// TIA Portal V17 export
// export: Created 2023-11-13T12:30:02.9222123Z, ExportSetting WithDefaults, DisplayName Totally Integrated Automation Portal, DisplayVersion V17, DisplayName TIA Portal Openness, DisplayVersion V17, DisplayName TIA Portal Version Control Interface, DisplayVersion V17, DisplayName STEP 7 Professional, DisplayVersion V17, DisplayName STEP 7 Safety, DisplayVersion V17, DisplayName WinCC Professional, DisplayVersion V17
FUNCTION_BLOCK "Motor"   // FB11, FBD
{ S7_Optimized_Access := 'TRUE' }
VERSION : 0.1
// stored: AutoNumber true, IsIECCheckEnabled false, IsRetainMemResEnabled false, MemoryReserve 100, SetENOAutomatically false, UDAEnableTagReadback false
   VAR_INPUT
      CON : Bool;
      COFF : Bool := 1;
      TagName : String[16];
      "PCS/PLC" : Bool;
      PCS_Auto : Bool;
      Ready : Bool;
      Running : Bool;
      STAITL : Bool := 1;
      PSTITL : Bool := 1;
      STPITL : Bool := 1;
      OPITL : Bool := 1;
      PRTITL : Bool := 1;
      FO { ExternalAccessible := 'False'; ExternalVisible := 'False'; ExternalWritable := 'False'} : Bool;   // First Out
      PHYFB : Bool := 1;
   END_VAR
   VAR_OUTPUT
      AVBL : Bool;
      ON : Bool;
      RUN : Bool;
      Start_PCS : Bool;
      Stop_PCS : Bool;
      Interlock_PCS : Bool;
      Screen : Bool;
   END_VAR
   VAR_IN_OUT
      Popup : "Popup_MtrOnOff";   // Common Popup Data
   END_VAR
   VAR
      "Local start" : Bool;
      "Local stop" : Bool;
      Remote : Bool;
      "Remote release" : Bool;
      Local : Bool;
      "Local release" : Bool;
      "Motor fault (electrically)" : Bool;
      "Feedback contactor" : Bool;
      Start : Bool;
      Stop : Bool;
      FDBCK : Bool;
      "Stop/ITL" : Bool;
      "Stop/Run" : Bool;
      IEC_Timer_Feedback_On { S7_SetPoint := 'True'} : TON_TIME;
      IEC_Timer_Feedback_Off { S7_SetPoint := 'True'} : TON_TIME;
      IEC_Timer_Feedback_Run { S7_SetPoint := 'True'} : TON_TIME;
      FDBCK_On { S7_SetPoint := 'True'} : Bool;
      FDBCK_Off { S7_SetPoint := 'True'} : Bool;
      FDBCK_Run { S7_SetPoint := 'True'} : Bool;
   END_VAR
   VAR RETAIN
      Param { ExternalAccessible := 'False'; ExternalVisible := 'False'; ExternalWritable := 'False'} : Struct   // Internal Parameters
         ReversingMotor { ExternalAccessible := 'False'; ExternalVisible := 'False'; ExternalWritable := 'False'; S7_SetPoint := 'True'} : Bool := False;   // 1:Enable Direction Select
         SpeedSelect { ExternalAccessible := 'False'; ExternalVisible := 'False'; ExternalWritable := 'False'; S7_SetPoint := 'True'} : Bool := False;   // 1:Enable Speed Select
         EN_FB_Forward { ExternalAccessible := 'False'; ExternalVisible := 'False'; ExternalWritable := 'False'; S7_SetPoint := 'True'} : Bool := true;   // 1:Enable FB_Forward
         EN_FB_Revsere { ExternalAccessible := 'False'; ExternalVisible := 'False'; ExternalWritable := 'False'; S7_SetPoint := 'True'} : Bool := true;   // 1:Enable FB_Reverse
         Disable_MCC_FLT { ExternalAccessible := 'False'; ExternalVisible := 'False'; ExternalWritable := 'False'; S7_SetPoint := 'True'} : Bool := false;   // 1:Disable MCC_FLT
         Disable_StartFLT { ExternalAccessible := 'False'; ExternalVisible := 'False'; ExternalWritable := 'False'; S7_SetPoint := 'True'} : Bool := false;   // 1:Disable StartFLT
         Disable_StopFLT { ExternalAccessible := 'False'; ExternalVisible := 'False'; ExternalWritable := 'False'; S7_SetPoint := 'True'} : Bool := false;   // 1:Disable StopFLT
         Disable_ForwardFLT { ExternalAccessible := 'False'; ExternalVisible := 'False'; ExternalWritable := 'False'; S7_SetPoint := 'True'} : Bool := false;   // 1:Disable ForwardFLT
         Disable_ReverseFLT { ExternalAccessible := 'False'; ExternalVisible := 'False'; ExternalWritable := 'False'; S7_SetPoint := 'True'} : Bool := false;   // 1:Disable ReverseFLT
         CMD_PulseWidth { ExternalAccessible := 'False'; ExternalVisible := 'False'; ExternalWritable := 'False'; S7_SetPoint := 'True'} : Time := t#2s;   // Command Pulse width
         WatchdogTime { ExternalAccessible := 'False'; ExternalVisible := 'False'; ExternalWritable := 'False'; S7_SetPoint := 'True'} : Array[0..5] of Real;   // Watchdog time for Fault detection
         Bumpless { ExternalAccessible := 'False'; ExternalVisible := 'False'; ExternalWritable := 'False'; S7_SetPoint := 'True'} : Bool := true;   // 1:Bumpless Switching to PLC Remote
         OpeBy2Step { ExternalAccessible := 'False'; ExternalVisible := 'False'; ExternalWritable := 'False'; S7_SetPoint := 'True'} : Bool := true;   // 1:2Step Operation
         PopupTime { ExternalAccessible := 'False'; ExternalVisible := 'False'; ExternalWritable := 'False'; S7_SetPoint := 'True'} : Time := T#60s;   // Time to close Confiramtion box
         TotalNoOfHMI { ExternalAccessible := 'False'; ExternalVisible := 'False'; ExternalWritable := 'False'; S7_SetPoint := 'True'} : Int := 1;   // Total Number of HMI
      END_STRUCT;
   END_VAR
   VAR
      icon : "icon_MtrOnOff";   // Icon Data
      HMI : "Popup_MtrOnOff";   // HMI Display Data
      ActiveHMI { ExternalAccessible := 'False'; ExternalVisible := 'False'; ExternalWritable := 'False'} : "Popup_MtrOnOff";   // Active HMI Data (Work Data)
      PassiveHMI { ExternalAccessible := 'False'; ExternalVisible := 'False'; ExternalWritable := 'False'} : "Popup_MtrOnOff";   // Passive HMI Object Code
      PopupCtrl { ExternalAccessible := 'False'; ExternalVisible := 'False'; ExternalWritable := 'False'} : Struct   // Popup Control Data
         Opened { ExternalAccessible := 'False'; ExternalVisible := 'False'; ExternalWritable := 'False'} : Bool;   // Popup is opened on the HMI
         Activate { ExternalAccessible := 'False'; ExternalVisible := 'False'; ExternalWritable := 'False'} : Bool;   // Any Operating on the HMI
         ValueChange { ExternalAccessible := 'False'; ExternalVisible := 'False'; ExternalWritable := 'False'} : Bool;   // Any Value is chaging on the HMI
         OperationBlocked { ExternalAccessible := 'False'; ExternalVisible := 'False'; ExternalWritable := 'False'} : Bool;   // Operation is blocked (inhibited)
         TagNameNotSame { ExternalAccessible := 'False'; ExternalVisible := 'False'; ExternalWritable := 'False'} : Bool;   // Tag name is not same with opened Popup on the HMI
      END_STRUCT;
      Modifying { ExternalAccessible := 'False'; ExternalVisible := 'False'; ExternalWritable := 'False'} : Struct   // Value is being modifyed on HMI
         AnyValue { ExternalAccessible := 'False'; ExternalVisible := 'False'; ExternalWritable := 'False'} : Bool;
         WatchdogTime_MccFLT { ExternalAccessible := 'False'; ExternalVisible := 'False'; ExternalWritable := 'False'} : Bool;
         WatchdogTime_StartFLT { ExternalAccessible := 'False'; ExternalVisible := 'False'; ExternalWritable := 'False'; S7_SetPoint := 'True'} : Bool;
         WatchdogTime_StopFLT { ExternalAccessible := 'False'; ExternalVisible := 'False'; ExternalWritable := 'False'; S7_SetPoint := 'True'} : Bool;
         WatchdogTime_ForwardFLT { ExternalAccessible := 'False'; ExternalVisible := 'False'; ExternalWritable := 'False'; S7_SetPoint := 'True'} : Bool;
         WatchdogTime_ReverseFLT { ExternalAccessible := 'False'; ExternalVisible := 'False'; ExternalWritable := 'False'; S7_SetPoint := 'True'} : Bool;
      END_STRUCT;
      previous { ExternalAccessible := 'False'; ExternalVisible := 'False'; ExternalWritable := 'False'} : Struct   // Previous Values
         WatchdogTime { ExternalAccessible := 'False'; ExternalVisible := 'False'; ExternalWritable := 'False'} : Array[0..5] of Real;
      END_STRUCT;
      Check { ExternalAccessible := 'False'; ExternalVisible := 'False'; ExternalWritable := 'False'} : Struct   // Check Value
         PBNo { ExternalAccessible := 'False'; ExternalVisible := 'False'; ExternalWritable := 'False'} : Int;
         WatchdogTime { ExternalAccessible := 'False'; ExternalVisible := 'False'; ExternalWritable := 'False'} : Real;
      END_STRUCT;
      HMI_PB { ExternalAccessible := 'False'; ExternalVisible := 'False'; ExternalWritable := 'False'} : Struct   // Push Buttons on Popup
         Remote { ExternalAccessible := 'False'; ExternalVisible := 'False'; ExternalWritable := 'False'} : Bool;
         Local { ExternalAccessible := 'False'; ExternalVisible := 'False'; ExternalWritable := 'False'} : Bool;
         Auto { ExternalAccessible := 'False'; ExternalVisible := 'False'; ExternalWritable := 'False'} : Bool;
         Manual { ExternalAccessible := 'False'; ExternalVisible := 'False'; ExternalWritable := 'False'} : Bool;
         Forward { ExternalAccessible := 'False'; ExternalVisible := 'False'; ExternalWritable := 'False'} : Bool;
         Reverse { ExternalAccessible := 'False'; ExternalVisible := 'False'; ExternalWritable := 'False'} : Bool;
         Speed1 { ExternalAccessible := 'False'; ExternalVisible := 'False'; ExternalWritable := 'False'} : Bool;
         Speed2 { ExternalAccessible := 'False'; ExternalVisible := 'False'; ExternalWritable := 'False'} : Bool;
         Start { ExternalAccessible := 'False'; ExternalVisible := 'False'; ExternalWritable := 'False'} : Bool;
         Stop { ExternalAccessible := 'False'; ExternalVisible := 'False'; ExternalWritable := 'False'} : Bool;
         ResetRT { ExternalAccessible := 'False'; ExternalVisible := 'False'; ExternalWritable := 'False'} : Bool;
         FO { ExternalAccessible := 'False'; ExternalVisible := 'False'; ExternalWritable := 'False'} : Bool;
      END_STRUCT;
      PLC_IN { ExternalAccessible := 'False'; ExternalVisible := 'False'; ExternalWritable := 'False'} : Struct   // PLC Signal operated on HMI
         Remote { ExternalAccessible := 'False'; ExternalVisible := 'False'; ExternalWritable := 'False'} : Bool;   // 0:Local / 1:Remote by PLC(HMI)
         Auto { ExternalAccessible := 'False'; ExternalVisible := 'False'; ExternalWritable := 'False'} : Bool;   // 0:Manual / 1:Auto by PLC(HMI)
         Start { ExternalAccessible := 'False'; ExternalVisible := 'False'; ExternalWritable := 'False'} : Bool;   // 1:Start by PLC(HMI)
         Stop { ExternalAccessible := 'False'; ExternalVisible := 'False'; ExternalWritable := 'False'} : Bool;   // 1: Stop by PLC(HMI)
         Reverse { ExternalAccessible := 'False'; ExternalVisible := 'False'; ExternalWritable := 'False'} : Bool;   // 0:Forward / 1:Reverse by PLC(HMI)
         Speed { ExternalAccessible := 'False'; ExternalVisible := 'False'; ExternalWritable := 'False'} : Bool;   // 0:Speed1 / 1:Speed2 by PLC(HMI)
      END_STRUCT;
      PBNo { ExternalAccessible := 'False'; ExternalVisible := 'False'; ExternalWritable := 'False'} : Int;   // Internal PBNo
      HMI_Operating { ExternalAccessible := 'False'; ExternalVisible := 'False'; ExternalWritable := 'False'} : Bool;   // Operating on HMI
      Popup_Open { ExternalAccessible := 'False'; ExternalVisible := 'False'; ExternalWritable := 'False'} : Bool;   // Any Popup is Opened
      Popup_Activate { ExternalAccessible := 'False'; ExternalVisible := 'False'; ExternalWritable := 'False'} : Bool;   // Any Popup is Activated
      Init { ExternalAccessible := 'False'; ExternalVisible := 'False'; ExternalWritable := 'False'} : Bool;
      ExternalReset { ExternalAccessible := 'False'; ExternalVisible := 'False'; ExternalWritable := 'False'} : Bool;   // External Reset
      Confirm { ExternalAccessible := 'False'; ExternalVisible := 'False'; ExternalWritable := 'False'} : Bool;   // Confirm Action
      Cancel { ExternalAccessible := 'False'; ExternalVisible := 'False'; ExternalWritable := 'False'} : Bool;   // Cancel Action
      CancelTimer { ExternalAccessible := 'False'; ExternalVisible := 'False'; ExternalWritable := 'False'} : Bool;   // Cancel Timer
      Enable { ExternalAccessible := 'False'; ExternalVisible := 'False'; ExternalWritable := 'False'} : Bool;   // 1:Enable Motor Operation
      Start_1 { ExternalAccessible := 'False'; ExternalVisible := 'False'; ExternalWritable := 'False'} : Bool;   // 1:Start Command ON
      Field_ForwardPLS { ExternalAccessible := 'False'; ExternalVisible := 'False'; ExternalWritable := 'False'} : Bool;   // Field Forward Pulse
      Field_ReversePLS { ExternalAccessible := 'False'; ExternalVisible := 'False'; ExternalWritable := 'False'} : Bool;   // Field Reverse Pulse
      SIM { ExternalAccessible := 'False'; ExternalVisible := 'False'; ExternalWritable := 'False'} : Bool;   // 1: SIM Mode (Automatic Answer)
      RT { ExternalAccessible := 'False'; ExternalVisible := 'False'; ExternalWritable := 'False'} : Struct   // RunTime
         hour { ExternalAccessible := 'False'; ExternalVisible := 'False'; ExternalWritable := 'False'} : DInt;
         min { ExternalAccessible := 'False'; ExternalVisible := 'False'; ExternalWritable := 'False'} : DInt;
         sec { ExternalAccessible := 'False'; ExternalVisible := 'False'; ExternalWritable := 'False'} : Int;
         ActSec { ExternalAccessible := 'False'; ExternalVisible := 'False'; ExternalWritable := 'False'} : USInt;
         Edge { ExternalAccessible := 'False'; ExternalVisible := 'False'; ExternalWritable := 'False'} : Bool;
         Reset { ExternalAccessible := 'False'; ExternalVisible := 'False'; ExternalWritable := 'False'} : Bool;
      END_STRUCT;
      Clear { ExternalAccessible := 'False'; ExternalVisible := 'False'; ExternalWritable := 'False'} : "Popup_MtrOnOff";   // for Clear Popup Data
      Edge { ExternalAccessible := 'False'; ExternalVisible := 'False'; ExternalWritable := 'False'} : Struct   // for Edging
         Remote { ExternalAccessible := 'False'; ExternalVisible := 'False'; ExternalWritable := 'False'} : Bool;
         Local { ExternalAccessible := 'False'; ExternalVisible := 'False'; ExternalWritable := 'False'} : Bool;
         Auto { ExternalAccessible := 'False'; ExternalVisible := 'False'; ExternalWritable := 'False'} : Bool;
         Manual { ExternalAccessible := 'False'; ExternalVisible := 'False'; ExternalWritable := 'False'} : Bool;
         Forward { ExternalAccessible := 'False'; ExternalVisible := 'False'; ExternalWritable := 'False'} : Bool;
         Reverse { ExternalAccessible := 'False'; ExternalVisible := 'False'; ExternalWritable := 'False'} : Bool;
         Speed1 { ExternalAccessible := 'False'; ExternalVisible := 'False'; ExternalWritable := 'False'} : Bool;
         Speed2 { ExternalAccessible := 'False'; ExternalVisible := 'False'; ExternalWritable := 'False'} : Bool;
         Start { ExternalAccessible := 'False'; ExternalVisible := 'False'; ExternalWritable := 'False'} : Bool;
         Stop { ExternalAccessible := 'False'; ExternalVisible := 'False'; ExternalWritable := 'False'} : Bool;
         HMI_Remote { ExternalAccessible := 'False'; ExternalVisible := 'False'; ExternalWritable := 'False'} : Bool;
         HMI_Local { ExternalAccessible := 'False'; ExternalVisible := 'False'; ExternalWritable := 'False'} : Bool;
         HMI_Auto { ExternalAccessible := 'False'; ExternalVisible := 'False'; ExternalWritable := 'False'} : Bool;
         HMI_Manual { ExternalAccessible := 'False'; ExternalVisible := 'False'; ExternalWritable := 'False'} : Bool;
         HMI_Forward { ExternalAccessible := 'False'; ExternalVisible := 'False'; ExternalWritable := 'False'} : Bool;
         HMI_Reverse { ExternalAccessible := 'False'; ExternalVisible := 'False'; ExternalWritable := 'False'} : Bool;
         HMI_Speed1 { ExternalAccessible := 'False'; ExternalVisible := 'False'; ExternalWritable := 'False'} : Bool;
         HMI_Speed2 { ExternalAccessible := 'False'; ExternalVisible := 'False'; ExternalWritable := 'False'} : Bool;
         PCS_Remote { ExternalAccessible := 'False'; ExternalVisible := 'False'; ExternalWritable := 'False'} : Bool;
         PCS_Local { ExternalAccessible := 'False'; ExternalVisible := 'False'; ExternalWritable := 'False'} : Bool;
         PCS_Auto { ExternalAccessible := 'False'; ExternalVisible := 'False'; ExternalWritable := 'False'} : Bool;
         PCS_Manual { ExternalAccessible := 'False'; ExternalVisible := 'False'; ExternalWritable := 'False'} : Bool;
         PCS_Forward { ExternalAccessible := 'False'; ExternalVisible := 'False'; ExternalWritable := 'False'} : Bool;
         PCS_Reverse { ExternalAccessible := 'False'; ExternalVisible := 'False'; ExternalWritable := 'False'} : Bool;
         PCS_Speed1 { ExternalAccessible := 'False'; ExternalVisible := 'False'; ExternalWritable := 'False'} : Bool;
         PCS_Speed2 { ExternalAccessible := 'False'; ExternalVisible := 'False'; ExternalWritable := 'False'} : Bool;
         PCS_Start { ExternalAccessible := 'False'; ExternalVisible := 'False'; ExternalWritable := 'False'} : Bool;
         PCS_Stop { ExternalAccessible := 'False'; ExternalVisible := 'False'; ExternalWritable := 'False'} : Bool;
         PLC_Remote { ExternalAccessible := 'False'; ExternalVisible := 'False'; ExternalWritable := 'False'} : Bool;
         PLC_Local { ExternalAccessible := 'False'; ExternalVisible := 'False'; ExternalWritable := 'False'} : Bool;
         PLC_Auto { ExternalAccessible := 'False'; ExternalVisible := 'False'; ExternalWritable := 'False'} : Bool;
         PLC_Manual { ExternalAccessible := 'False'; ExternalVisible := 'False'; ExternalWritable := 'False'} : Bool;
         PLC_Forward { ExternalAccessible := 'False'; ExternalVisible := 'False'; ExternalWritable := 'False'} : Bool;
         PLC_Reverse { ExternalAccessible := 'False'; ExternalVisible := 'False'; ExternalWritable := 'False'} : Bool;
         PLC_Speed1 { ExternalAccessible := 'False'; ExternalVisible := 'False'; ExternalWritable := 'False'} : Bool;
         PLC_Speed2 { ExternalAccessible := 'False'; ExternalVisible := 'False'; ExternalWritable := 'False'} : Bool;
         PLC_Start { ExternalAccessible := 'False'; ExternalVisible := 'False'; ExternalWritable := 'False'} : Bool;
         PLC_Stop { ExternalAccessible := 'False'; ExternalVisible := 'False'; ExternalWritable := 'False'} : Bool;
         Auto_Start { ExternalAccessible := 'False'; ExternalVisible := 'False'; ExternalWritable := 'False'} : Bool;
         Auto_Stop { ExternalAccessible := 'False'; ExternalVisible := 'False'; ExternalWritable := 'False'} : Bool;
         Auto_Forward { ExternalAccessible := 'False'; ExternalVisible := 'False'; ExternalWritable := 'False'} : Bool;
         Auto_Reverse { ExternalAccessible := 'False'; ExternalVisible := 'False'; ExternalWritable := 'False'} : Bool;
         Auto_Speed1 { ExternalAccessible := 'False'; ExternalVisible := 'False'; ExternalWritable := 'False'} : Bool;
         Auto_Speed2 { ExternalAccessible := 'False'; ExternalVisible := 'False'; ExternalWritable := 'False'} : Bool;
         AutoREQ { ExternalAccessible := 'False'; ExternalVisible := 'False'; ExternalWritable := 'False'} : Bool;
         ManualREQ { ExternalAccessible := 'False'; ExternalVisible := 'False'; ExternalWritable := 'False'} : Bool;
         Field_Forward { ExternalAccessible := 'False'; ExternalVisible := 'False'; ExternalWritable := 'False'} : Bool;
         Field_Reverse { ExternalAccessible := 'False'; ExternalVisible := 'False'; ExternalWritable := 'False'} : Bool;
         Field_Stop { ExternalAccessible := 'False'; ExternalVisible := 'False'; ExternalWritable := 'False'} : Bool;
         Confirm { ExternalAccessible := 'False'; ExternalVisible := 'False'; ExternalWritable := 'False'} : Bool;
         Cancel1 { ExternalAccessible := 'False'; ExternalVisible := 'False'; ExternalWritable := 'False'} : Bool;
         Cancel2 { ExternalAccessible := 'False'; ExternalVisible := 'False'; ExternalWritable := 'False'} : Bool;
         Cancel3 { ExternalAccessible := 'False'; ExternalVisible := 'False'; ExternalWritable := 'False'} : Bool;
         ModifyValue { ExternalAccessible := 'False'; ExternalVisible := 'False'; ExternalWritable := 'False'} : Bool;
      END_STRUCT;
      TP_PLC_Start { ExternalAccessible := 'False'; ExternalVisible := 'False'; ExternalWritable := 'False'} : TP_TIME;   // PLC Start Pulse Timer
      TP_PLC_Stop { ExternalAccessible := 'False'; ExternalVisible := 'False'; ExternalWritable := 'False'} : TP_TIME;   // PLC Stop Pulse Timer
      TP_CMD_FwdStart { ExternalAccessible := 'False'; ExternalVisible := 'False'; ExternalWritable := 'False'} : TP_TIME;   // Forward Start Command Pulse Timer
      TP_CMD_RvsStart { ExternalAccessible := 'False'; ExternalVisible := 'False'; ExternalWritable := 'False'} : TP_TIME;   // Reverse Start Command Pulse Timer
      TP_CMD_Stop { ExternalAccessible := 'False'; ExternalVisible := 'False'; ExternalWritable := 'False'} : TP_TIME;   // Stop Command Pulse Timer
      TON_MCC_FLT { ExternalAccessible := 'False'; ExternalVisible := 'False'; ExternalWritable := 'False'} : TON_TIME;   // MCC Fault Delay Timer
      TON_StartFLT { ExternalAccessible := 'False'; ExternalVisible := 'False'; ExternalWritable := 'False'} : TON_TIME;   // Start Fault Delay Timer
      TON_StopFLT { ExternalAccessible := 'False'; ExternalVisible := 'False'; ExternalWritable := 'False'} : TON_TIME;   // Stop Fault Delay Timer
      TON_ForwardFLT { ExternalAccessible := 'False'; ExternalVisible := 'False'; ExternalWritable := 'False'} : TON_TIME;   // Forward Fault Delay Timer
      TON_ReverseFLT { ExternalAccessible := 'False'; ExternalVisible := 'False'; ExternalWritable := 'False'} : TON_TIME;   // Reverse Fault Delay Timer
      TON_SIMON_Start { ExternalAccessible := 'False'; ExternalVisible := 'False'; ExternalWritable := 'False'} : TON_TIME;   // SIMON Start On-Delay Timer
      TP_SIMON_Stop { ExternalAccessible := 'False'; ExternalVisible := 'False'; ExternalWritable := 'False'} : TP_TIME;   // SIMON Stop Pulse Timer
      TON_Popup { ExternalAccessible := 'False'; ExternalVisible := 'False'; ExternalWritable := 'False'} : TON_TIME;   // Confirmation Popup Check Timer
      TP_Screen { ExternalAccessible := 'False'; ExternalVisible := 'False'; ExternalWritable := 'False'} : TP_TIME;   // Screen Pulse Timer
      TagComment { S7_SetPoint := 'True'} : String[32];
      PCS_Operation : Bool;
      Auto : Bool;
      Permit : Bool;
      Interlock : Bool;
      NonService : Bool;
      Fault : Bool;
      Speed : Bool;
      StartFLT : Bool;
      StopFLT : Bool;
      ForwardFLT : Bool;
      ReverseFLT : Bool;
      FaultReset : Bool;
      MCC_FLT : Bool;
      Reverse : Bool;
      CMD_Fwd { ExternalAccessible := 'False'; ExternalVisible := 'False'; ExternalWritable := 'False'} : Bool;   // 1: Forward Start Command
      CMD_Rvs { ExternalAccessible := 'False'; ExternalVisible := 'False'; ExternalWritable := 'False'} : Bool;   // 1: Reverse Start Command
      CMD_Stop { ExternalAccessible := 'False'; ExternalVisible := 'False'; ExternalWritable := 'False'} : Bool;   // 1: Stop Command
   END_VAR
   VAR_TEMP
      bTemp : Bool;   // Temporary bit
      Debug : Bool;
      dTemp : DInt;
      rTemp : Real;
      FB_FWD : Bool;   // Motor Forward running Status
      FB_RVS : Bool;   // Motor Reverse running Status
      Disable_FaultCheck : Bool;
      PT_MccFLT : Time;   // Watchdog time for Fault detection
      PT_StartFLT : Time;
      PT_StopFLT : Time;
      PT_ForwardFLT : Time;
      PT_ReverseFLT : Time;
      PT_SIMON : Time;
      No : Int;
      "Return" : Int;
      DTL : DTL;
   END_VAR
   VAR CONSTANT
      Local_PBNo : Int := 10;
      Remote_PBNo : Int := 11;
      Manual_PBNo : Int := 20;
      Auto_PBNo : Int := 21;
      Forward_PBNo : Int := 30;
      Reverse_PBNo : Int := 31;
      Speed1_PBNo : Int := 40;
      Speed2_PBNo : Int := 41;
      Stop_PBNo : Int := 50;
      Start_PBNo : Int := 51;
      ResetRT_PBNo : Int := 140;
      FO_PBNo : Int := 520;
      ValueChange_Popup : Int := 300;
   END_VAR
   // Param.WatchdogTime[0] := 0.0;
   // Param.WatchdogTime[1..5] := 10.0;
   VAR_TEMP   // added for the SCL form of the ladder/FBD networks
      _w1 : Bool;
      _w2 : Bool;
      _w3 : Bool;
      _w4 : Bool;
      _w5 : Bool;
      _w6 : Bool;
      _w7 : Bool;
      _w8 : Bool;
      _w9 : Bool;
   END_VAR
BEGIN

REGION Network 2: ----- Preperation ------------------------------------------------------------------------------------------------------------------------------------------------------------------------
END_REGION

REGION Network 3 (SCL): Parameter Set
   ////  Parameters which are fixed at the moment. //////////////////////////////////  

   // Start/Stop Command Pulse width     
   #Param.CMD_PulseWidth := t#3s;

   //Disable Fault 
   #Param.Disable_MCC_FLT := false;
   #Param.Disable_StartFLT := false;
   #Param.Disable_StopFLT := false;
   #Param.Disable_ForwardFLT := false;
   #Param.Disable_ReverseFLT := false;

   // Two Step Operation (True=Two Step, this parameter have to be true.)
   #Param.OpeBy2Step := true;


   //// Parameters which are common for all Library FBs. ////////////////////////////

   //  Confirm Button is disappeared after PopupTime. (Default=60s)  
   #Param.PopupTime := "HMI".Param.PopupTime;

   // Total No of Touch Panels which is connected to the CPU.
   // 1 <= "HMI".Param.TotalNoOfHMI <=10 , if not CPU stops
   #Param.TotalNoOfHMI := "HMI".Param.TotalNoOfHMI;
END_REGION

REGION Network 4 (SCL): Popup Screen Operation
   IF #Popup.TagName = #TagName THEN

           //Get Value when Popup Open (First Scan Action When Popup Opened)
           IF #PopupCtrl.Opened = false THEN
               #Popup.PBNo := #ActiveHMI.PBNo;
               #Popup.WatchdogTime := #ActiveHMI.WatchdogTime;
           END_IF;
           #PopupCtrl.Opened := true;

           //Any Value Change on this HMI ?
           IF #Popup.WatchdogTime[0]<>#previous.WatchdogTime[0] OR #Popup.WatchdogTime[1]<>#previous.WatchdogTime[1] OR //Any Value change ?
               #Popup.WatchdogTime[2]<>#previous.WatchdogTime[2] OR #Popup.WatchdogTime[3]<>#previous.WatchdogTime[3] OR
               #Popup.WatchdogTime[4]<>#previous.WatchdogTime[4] OR #Popup.WatchdogTime[5]<>#previous.WatchdogTime[5] THEN
               #PopupCtrl.ValueChange := true;
           ELSE
               #PopupCtrl.ValueChange := false;
           END_IF;

           //Case: All HMI is Deactivated, and Check the HMI Activated or not.
           IF #HMI_Operating = false THEN
               IF #Popup.PBNo > 0 OR #PopupCtrl.ValueChange = true THEN //Any Opeation on the HMI ?
                   #PopupCtrl.Activate := true;
               END_IF;
           END_IF;
           //Case: the HMI is being Activated (under Operation)
           IF #PopupCtrl.Activate = true THEN
               IF #Confirm = true OR #Cancel = true THEN
                   #PopupCtrl.Activate := false;
               ELSE
                   IF #ActiveHMI.PBNo<>#Popup.PBNo THEN #ActiveHMI.PBNo:=#Popup.PBNo;END_IF;
                   IF #ActiveHMI.WatchdogTime[0]<>#Popup.WatchdogTime[0] THEN #ActiveHMI.WatchdogTime[0]:=#Popup.WatchdogTime[0]; END_IF;
                   IF #ActiveHMI.WatchdogTime[1]<>#Popup.WatchdogTime[1] THEN #ActiveHMI.WatchdogTime[1]:=#Popup.WatchdogTime[1]; END_IF;
                   IF #ActiveHMI.WatchdogTime[2]<>#Popup.WatchdogTime[2] THEN #ActiveHMI.WatchdogTime[2]:=#Popup.WatchdogTime[2]; END_IF;
                   IF #ActiveHMI.WatchdogTime[3]<>#Popup.WatchdogTime[3] THEN #ActiveHMI.WatchdogTime[3]:=#Popup.WatchdogTime[3]; END_IF;
                   IF #ActiveHMI.WatchdogTime[4]<>#Popup.WatchdogTime[4] THEN #ActiveHMI.WatchdogTime[4]:=#Popup.WatchdogTime[4]; END_IF;
                   IF #ActiveHMI.WatchdogTime[5]<>#Popup.WatchdogTime[5] THEN #ActiveHMI.WatchdogTime[5]:=#Popup.WatchdogTime[5]; END_IF;
               END_IF;
           ELSE
               IF #Popup.WatchdogTime[0]<>#Param.WatchdogTime[0] THEN #Popup.WatchdogTime[0]:=#Param.WatchdogTime[0]; END_IF;
               IF #Popup.WatchdogTime[1]<>#Param.WatchdogTime[1] THEN #Popup.WatchdogTime[1]:=#Param.WatchdogTime[1]; END_IF;
               IF #Popup.WatchdogTime[2]<>#Param.WatchdogTime[2] THEN #Popup.WatchdogTime[2]:=#Param.WatchdogTime[2]; END_IF;
               IF #Popup.WatchdogTime[3]<>#Param.WatchdogTime[3] THEN #Popup.WatchdogTime[3]:=#Param.WatchdogTime[3]; END_IF;
               IF #Popup.WatchdogTime[4]<>#Param.WatchdogTime[4] THEN #Popup.WatchdogTime[4]:=#Param.WatchdogTime[4]; END_IF;
               IF #Popup.WatchdogTime[5]<>#Param.WatchdogTime[5] THEN #Popup.WatchdogTime[5]:=#Param.WatchdogTime[5]; END_IF;

           END_IF;
           #PopupCtrl.TagNameNotSame := false;

       ELSE
           #PopupCtrl.Opened := false;
           #PopupCtrl.Activate := false;
           #PopupCtrl.ValueChange := false;
           IF #PopupCtrl.TagNameNotSame = false THEN
               #ActiveHMI.PBNo := 0;
               #PBNo := 0;
               #Popup := #Clear;
           END_IF;
           #PopupCtrl.TagNameNotSame := true;

       END_IF;
END_REGION

REGION Network 5: ----------- Common HMI Operation, Trigger Action ------------------------------------------------------------------------------------------------------------------
END_REGION

REGION Network 6: PBNo Operation (First Operation) /If PBNo>-10, It means First PB is pushed.
   // PBNo=10 : Local PB, PBNo=11 : Remote PB
   // PBNo=20 : Manual PB, PBNo=21 : Auto PB
   // PBNo=30 : Reverse PB, PBNo=31 : Forard PB
   // PBNo=40 : Speed1, PBNo=41 : Speed2 PB
   // PBNo=50 : Stop PB, PBNo=51 : Start PB
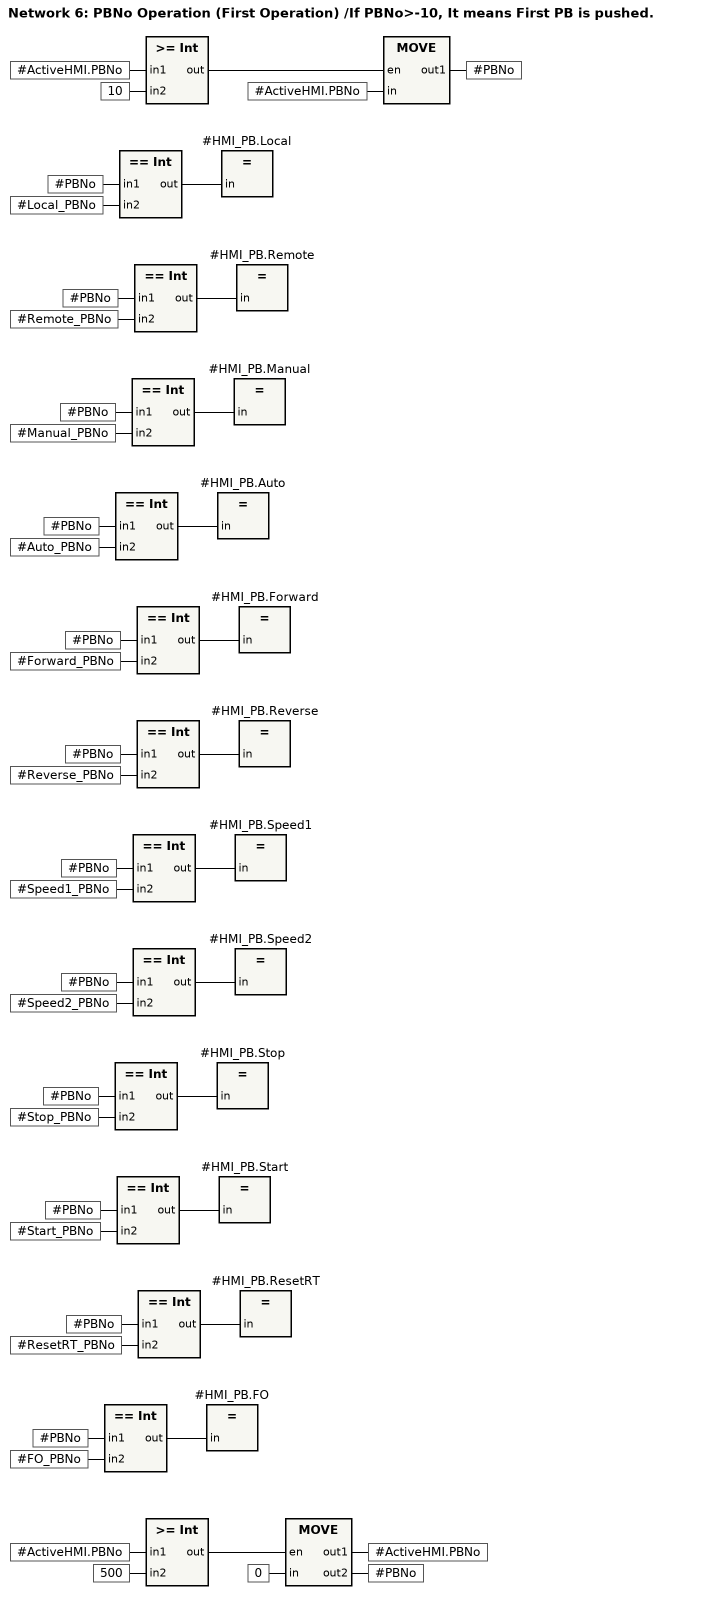
   IF #ActiveHMI.PBNo >= 10 THEN #PBNo := #ActiveHMI.PBNo; END_IF;
   #HMI_PB.Local := #PBNo = #Local_PBNo;
   #HMI_PB.Remote := #PBNo = #Remote_PBNo;
   #HMI_PB.Manual := #PBNo = #Manual_PBNo;
   #HMI_PB.Auto := #PBNo = #Auto_PBNo;
   #HMI_PB.Forward := #PBNo = #Forward_PBNo;
   #HMI_PB.Reverse := #PBNo = #Reverse_PBNo;
   #HMI_PB.Speed1 := #PBNo = #Speed1_PBNo;
   #HMI_PB.Speed2 := #PBNo = #Speed2_PBNo;
   #HMI_PB.Stop := #PBNo = #Stop_PBNo;
   #HMI_PB.Start := #PBNo = #Start_PBNo;
   #HMI_PB.ResetRT := #PBNo = #ResetRT_PBNo;
   #HMI_PB.FO := #PBNo = #FO_PBNo;
   IF #ActiveHMI.PBNo >= 500 THEN
       #ActiveHMI.PBNo := 0;
       #PBNo := 0;
   END_IF;
END_REGION

REGION Network 7: Value is being modified on HMI (not used)
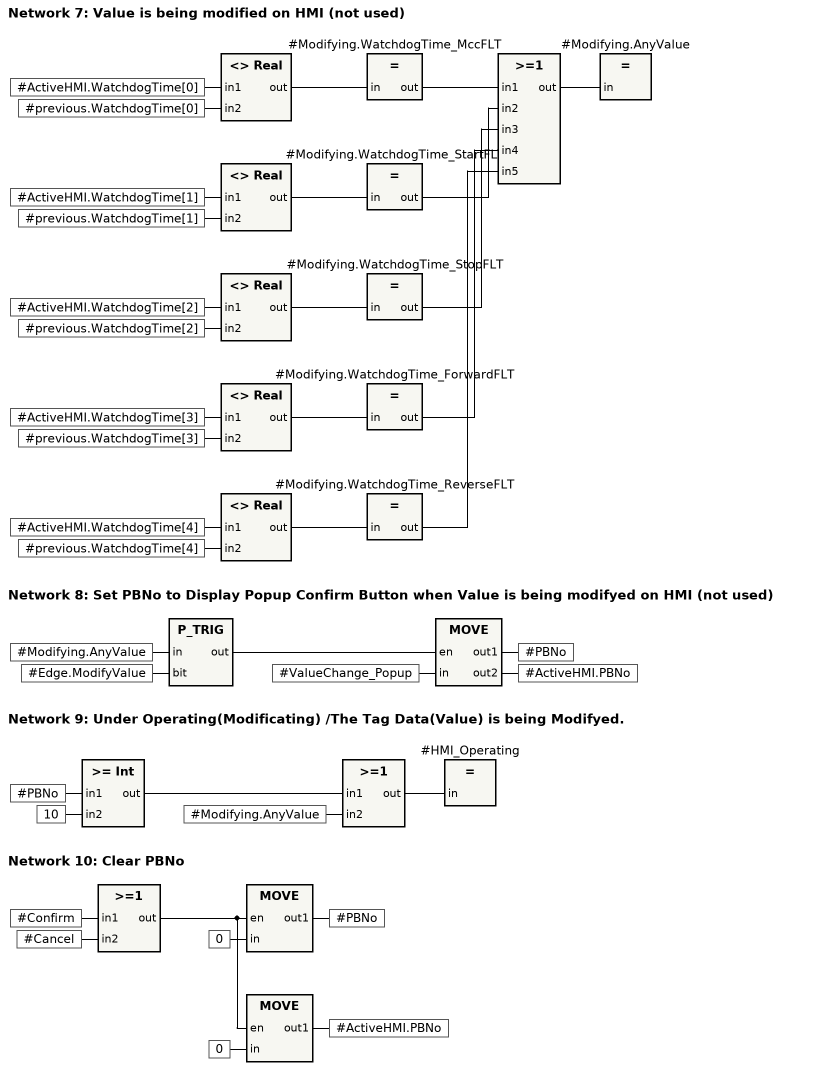
   #Modifying.WatchdogTime_MccFLT := #ActiveHMI.WatchdogTime[0] <> #previous.WatchdogTime[0];
   #Modifying.WatchdogTime_StartFLT := #ActiveHMI.WatchdogTime[1] <> #previous.WatchdogTime[1];
   #Modifying.WatchdogTime_StopFLT := #ActiveHMI.WatchdogTime[2] <> #previous.WatchdogTime[2];
   #Modifying.WatchdogTime_ForwardFLT := #ActiveHMI.WatchdogTime[3] <> #previous.WatchdogTime[3];
   #Modifying.WatchdogTime_ReverseFLT := #ActiveHMI.WatchdogTime[4] <> #previous.WatchdogTime[4];
   #Modifying.AnyValue := #Modifying.WatchdogTime_MccFLT OR #Modifying.WatchdogTime_StartFLT OR #Modifying.WatchdogTime_StopFLT OR #Modifying.WatchdogTime_ForwardFLT OR #Modifying.WatchdogTime_ReverseFLT;
END_REGION

REGION Network 8: Set PBNo to Display Popup Confirm Button when Value is being modifyed on HMI (not used)
   #_w1 := #Modifying.AnyValue AND NOT #Edge.ModifyValue;   // rising edge
   #Edge.ModifyValue := #Modifying.AnyValue;
   IF #_w1 THEN
       #PBNo := #ValueChange_Popup;
       #ActiveHMI.PBNo := #ValueChange_Popup;
   END_IF;
END_REGION

REGION Network 9: Under Operating(Modificating) /The Tag Data(Value) is being Modifyed.
   #HMI_Operating := (#PBNo >= 10) OR #Modifying.AnyValue;
END_REGION

REGION Network 10: Clear PBNo
   IF #Confirm OR #Cancel THEN
       #PBNo := 0;
       #ActiveHMI.PBNo := 0;
   END_IF;
END_REGION

REGION Network 11: Watchdog(60sec Timer) for Cancel Operation /Operation is canceled after Watchdog Time
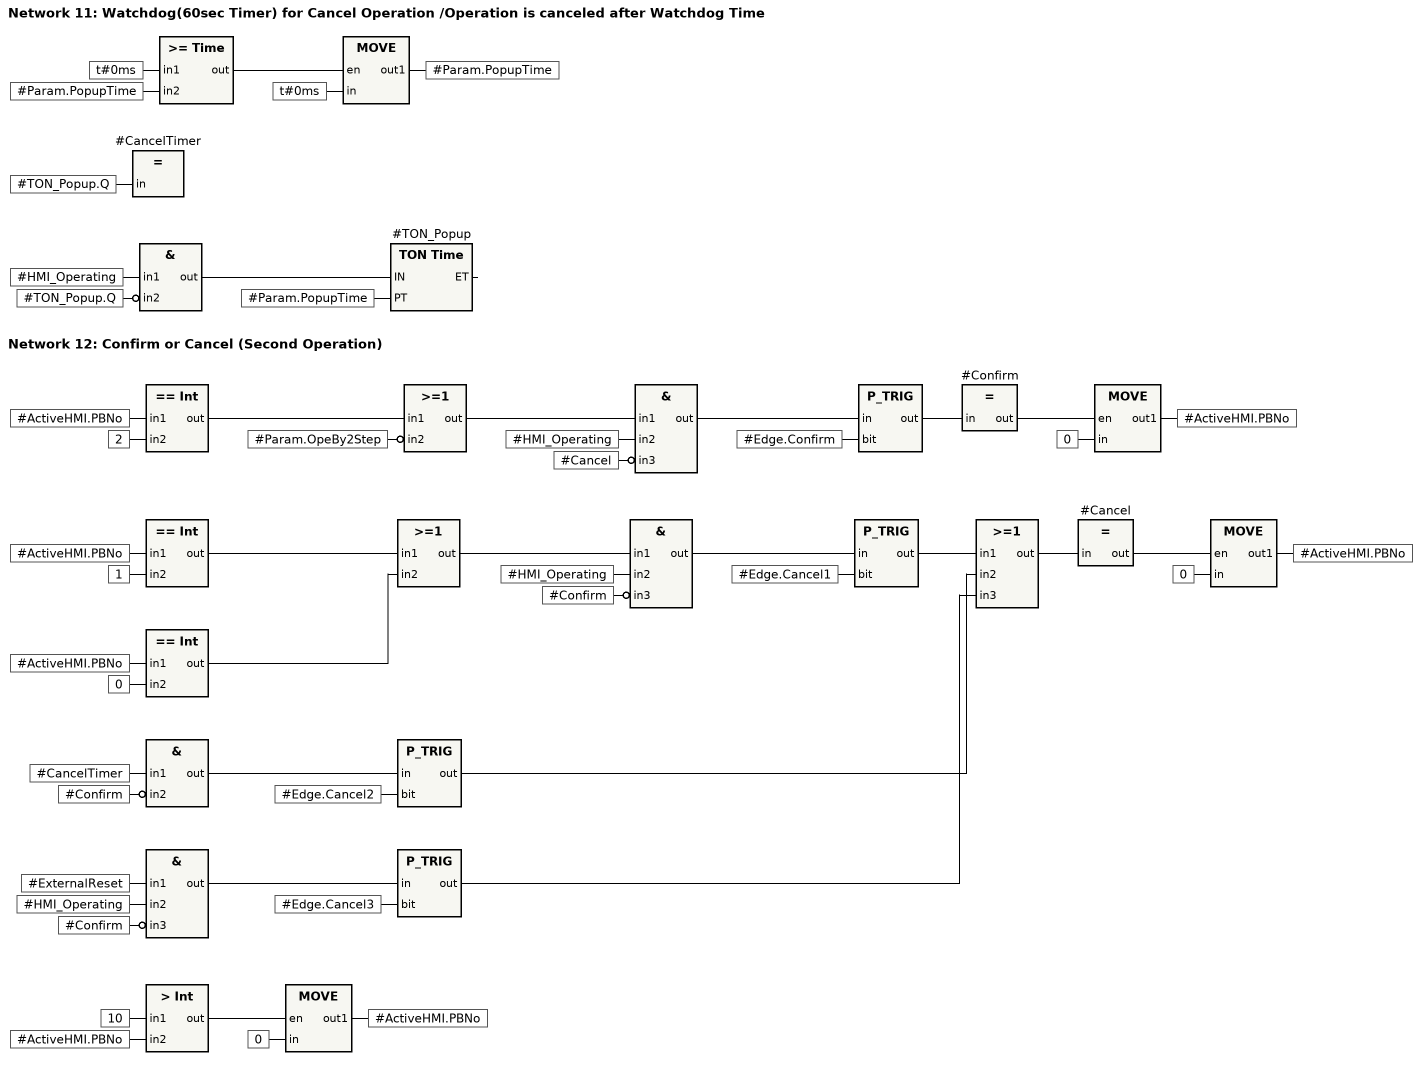
   IF t#0ms >= #Param.PopupTime THEN #Param.PopupTime := t#0ms; END_IF;
   #CancelTimer := #TON_Popup.Q;
   #TON_Popup(IN := #HMI_Operating AND NOT #TON_Popup.Q, PT := #Param.PopupTime);   // TON
END_REGION

REGION Network 12: Confirm or Cancel (Second Operation)
   // OpeBy2Step=1 : 2Step Operation / ExecutePB&CancelPB is necessary on HMI
   // OpeBy2Step=0 : 2Step Operation / ExecutePB&CancelPB is necessary on HMI
   // PBNo= 1:Cancel, 2:Confirm
   #_w1 := ((#ActiveHMI.PBNo = 2) OR NOT #Param.OpeBy2Step) AND #HMI_Operating AND NOT #Cancel;
   #_w2 := #_w1 AND NOT #Edge.Confirm;   // rising edge
   #Edge.Confirm := #_w1;
   #Confirm := #_w2;
   IF #_w2 THEN #ActiveHMI.PBNo := 0; END_IF;
   #_w3 := ((#ActiveHMI.PBNo = 1) OR (#ActiveHMI.PBNo = 0)) AND #HMI_Operating AND NOT #Confirm;
   #_w4 := #_w3 AND NOT #Edge.Cancel1;   // rising edge
   #Edge.Cancel1 := #_w3;
   #_w5 := #CancelTimer AND NOT #Confirm;
   #_w6 := #_w5 AND NOT #Edge.Cancel2;   // rising edge
   #Edge.Cancel2 := #_w5;
   #_w7 := #ExternalReset AND #HMI_Operating AND NOT #Confirm;
   #_w8 := #_w7 AND NOT #Edge.Cancel3;   // rising edge
   #Edge.Cancel3 := #_w7;
   #Cancel := #_w4 OR #_w6 OR #_w8;
   IF #Cancel THEN #ActiveHMI.PBNo := 0; END_IF;
   IF 10 > #ActiveHMI.PBNo THEN #ActiveHMI.PBNo := 0; END_IF;
END_REGION

REGION Network 13: ----------- PLC Action --------------------------------------------------------------------------------------------------------------------------------------------------------------------
END_REGION

REGION Network 14: HMI Push Button Check ---> PLC Request
   // The following PBNo is set when PB is pushed on HMI Pupupg Screen
   // PBNo=10 : Local PB is pushed.
   // PBNo=11 : Remote PB is pushed.
   // PBNo=20 : Manual PB is pushed.
   // PBNo=21 : Auto PB is pushed.
   // PBNo=30 : Reverse PB is pushed.
   // PBNo=31 : Forward PB is pushed.
   // PBNo=40 : Speed1 PB is pushed.
   // PBNo=41 : Speed2 PB is pushed.
   // PBNo=50 : Stop PB is pushed.
   // PBNo=51 : Start PB is pushed.
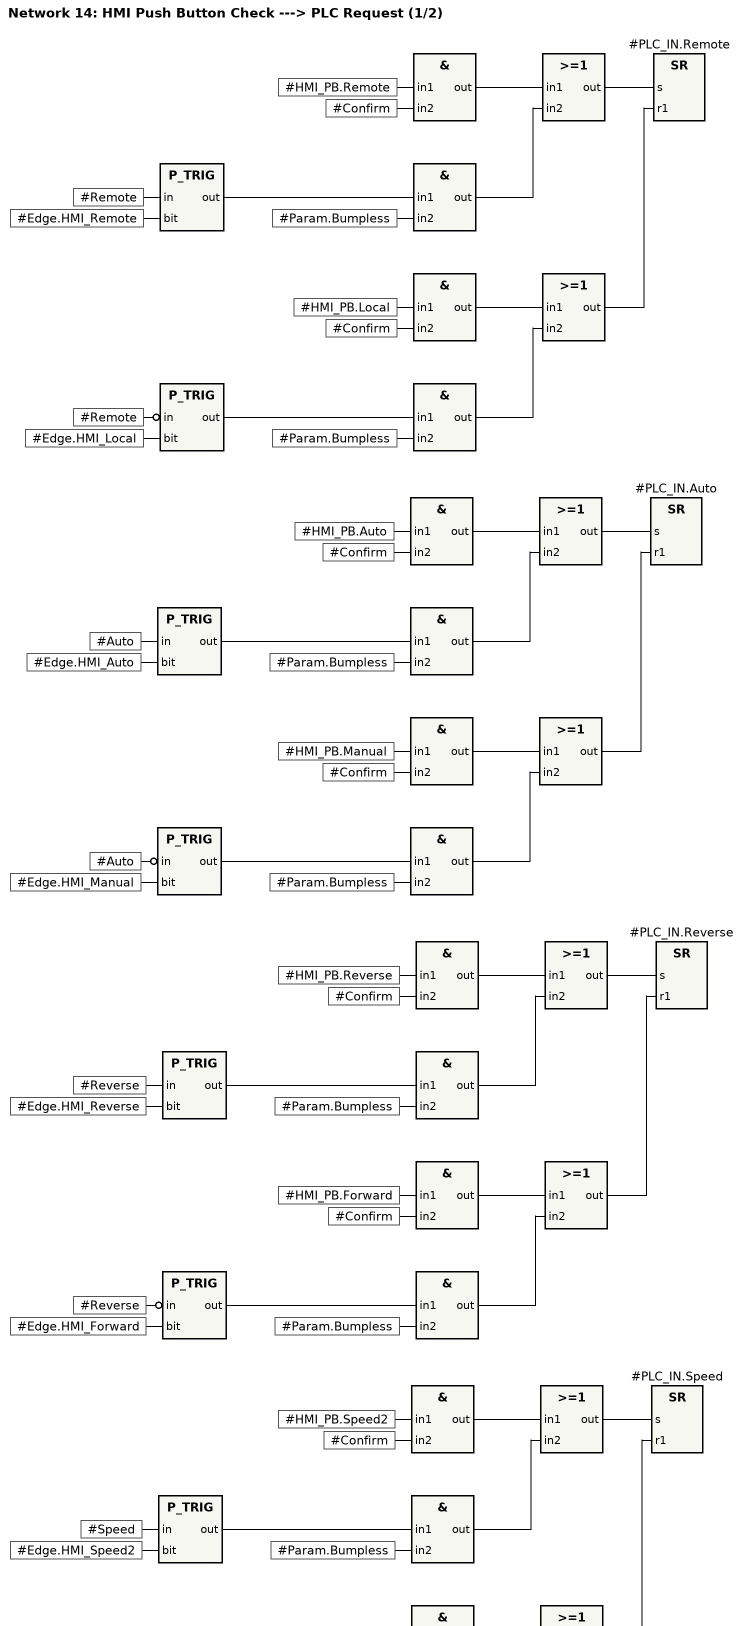
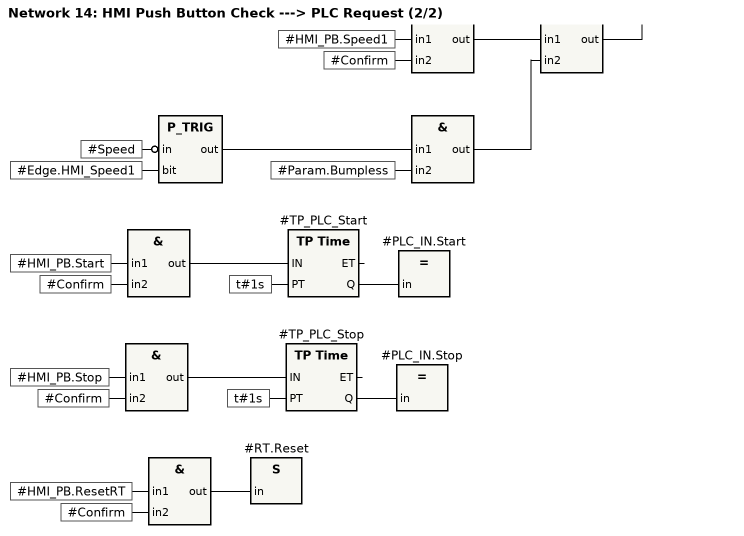
   #_w1 := #Remote AND NOT #Edge.HMI_Remote;   // rising edge
   #Edge.HMI_Remote := #Remote;
   #_w2 := NOT #Remote AND NOT #Edge.HMI_Local;   // rising edge
   #Edge.HMI_Local := NOT #Remote;
   IF (#HMI_PB.Remote AND #Confirm) OR (#_w1 AND #Param.Bumpless) THEN
       #PLC_IN.Remote := TRUE;   // SR flip-flop
   END_IF;
   IF (#HMI_PB.Local AND #Confirm) OR (#_w2 AND #Param.Bumpless) THEN #PLC_IN.Remote := FALSE; END_IF;
   #_w3 := #Auto AND NOT #Edge.HMI_Auto;   // rising edge
   #Edge.HMI_Auto := #Auto;
   #_w4 := NOT #Auto AND NOT #Edge.HMI_Manual;   // rising edge
   #Edge.HMI_Manual := NOT #Auto;
   IF (#HMI_PB.Auto AND #Confirm) OR (#_w3 AND #Param.Bumpless) THEN
       #PLC_IN.Auto := TRUE;   // SR flip-flop
   END_IF;
   IF (#HMI_PB.Manual AND #Confirm) OR (#_w4 AND #Param.Bumpless) THEN #PLC_IN.Auto := FALSE; END_IF;
   #_w5 := #Reverse AND NOT #Edge.HMI_Reverse;   // rising edge
   #Edge.HMI_Reverse := #Reverse;
   #_w6 := NOT #Reverse AND NOT #Edge.HMI_Forward;   // rising edge
   #Edge.HMI_Forward := NOT #Reverse;
   IF (#HMI_PB.Reverse AND #Confirm) OR (#_w5 AND #Param.Bumpless) THEN
       #PLC_IN.Reverse := TRUE;   // SR flip-flop
   END_IF;
   IF (#HMI_PB.Forward AND #Confirm) OR (#_w6 AND #Param.Bumpless) THEN #PLC_IN.Reverse := FALSE; END_IF;
   #_w7 := #Speed AND NOT #Edge.HMI_Speed2;   // rising edge
   #Edge.HMI_Speed2 := #Speed;
   #_w8 := NOT #Speed AND NOT #Edge.HMI_Speed1;   // rising edge
   #Edge.HMI_Speed1 := NOT #Speed;
   IF (#HMI_PB.Speed2 AND #Confirm) OR (#_w7 AND #Param.Bumpless) THEN
       #PLC_IN.Speed := TRUE;   // SR flip-flop
   END_IF;
   IF (#HMI_PB.Speed1 AND #Confirm) OR (#_w8 AND #Param.Bumpless) THEN #PLC_IN.Speed := FALSE; END_IF;
   #TP_PLC_Start(IN := #HMI_PB.Start AND #Confirm, PT := t#1s);   // TP
   #PLC_IN.Start := #TP_PLC_Start.Q;
   #TP_PLC_Stop(IN := #HMI_PB.Stop AND #Confirm, PT := t#1s);   // TP
   #PLC_IN.Stop := #TP_PLC_Stop.Q;
   IF #HMI_PB.ResetRT AND #Confirm THEN #RT.Reset := TRUE; END_IF;
END_REGION

REGION Network 15: ----------- Watchdog Time -----------------------------------------------------------------------------------------------------------------------------------------------------------------
END_REGION

REGION Network 16: WatchdogTime[0] for MccFLT
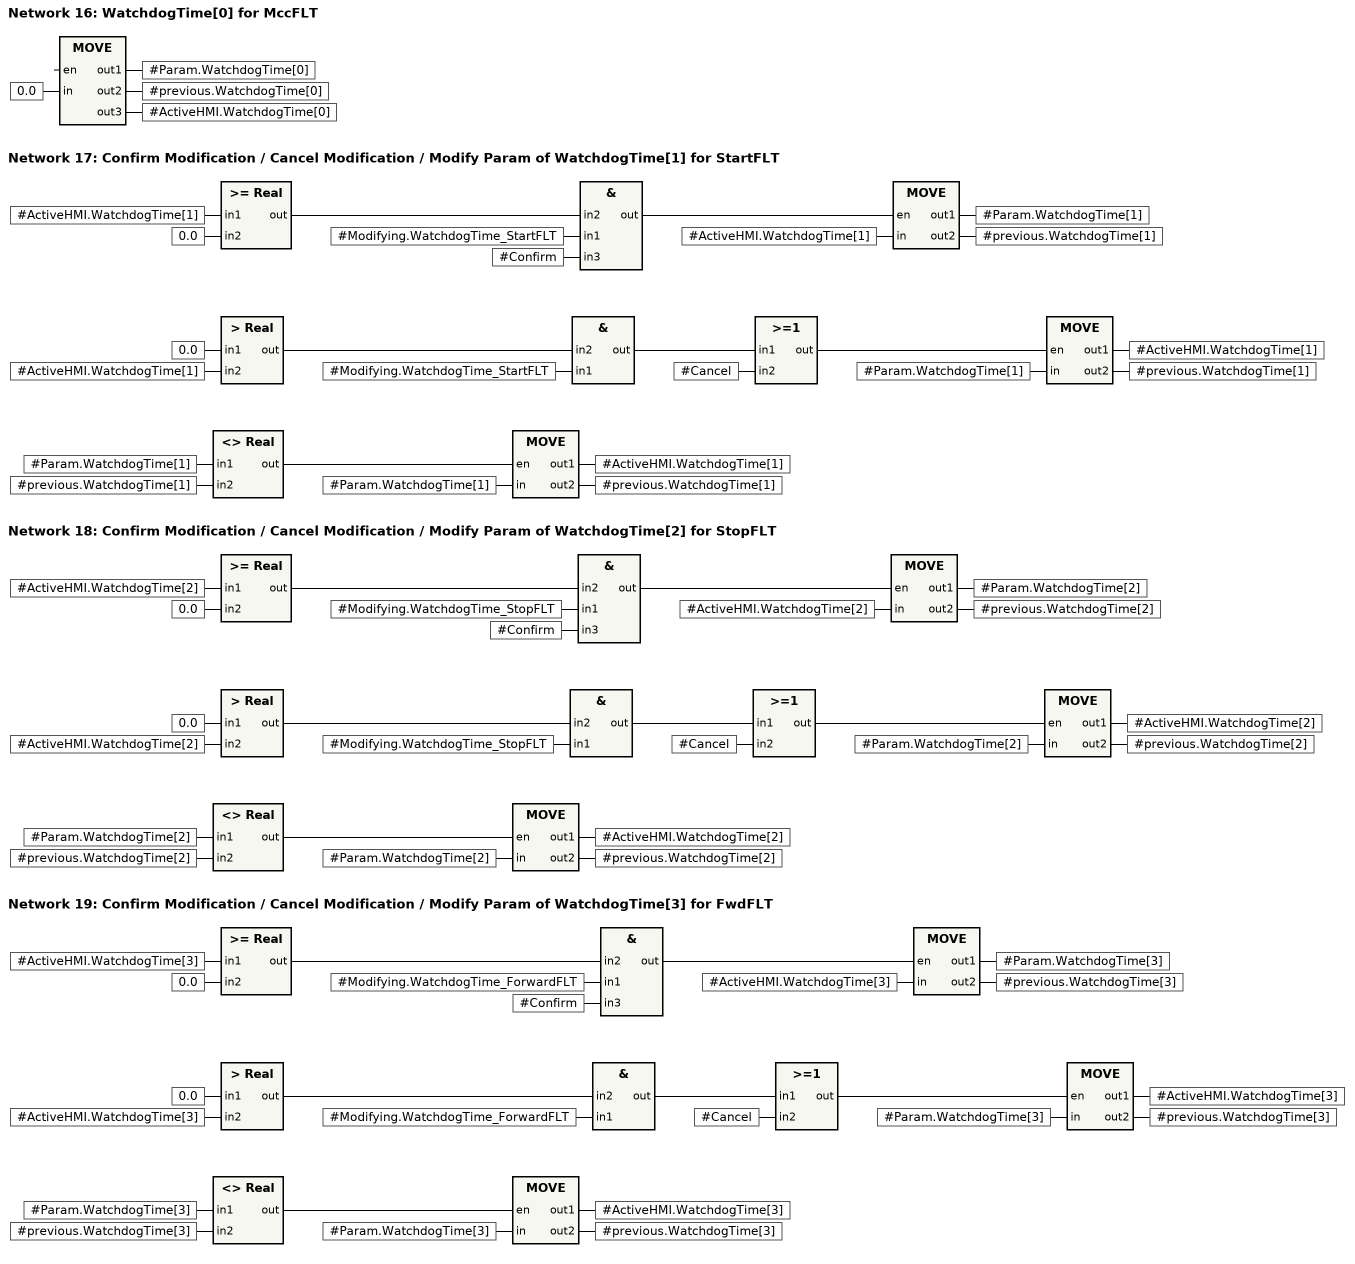
   #Param.WatchdogTime[0] := 0.0;
   #previous.WatchdogTime[0] := 0.0;
   #ActiveHMI.WatchdogTime[0] := 0.0;
END_REGION

REGION Network 17: Confirm Modification / Cancel Modification / Modify Param of WatchdogTime[1] for StartFLT
   IF (#ActiveHMI.WatchdogTime[1] >= 0.0) AND #Modifying.WatchdogTime_StartFLT AND #Confirm THEN
       #Param.WatchdogTime[1] := #ActiveHMI.WatchdogTime[1];
       #previous.WatchdogTime[1] := #ActiveHMI.WatchdogTime[1];
   END_IF;
   IF ((0.0 > #ActiveHMI.WatchdogTime[1]) AND #Modifying.WatchdogTime_StartFLT) OR #Cancel THEN
       #ActiveHMI.WatchdogTime[1] := #Param.WatchdogTime[1];
       #previous.WatchdogTime[1] := #Param.WatchdogTime[1];
   END_IF;
   IF #Param.WatchdogTime[1] <> #previous.WatchdogTime[1] THEN
       #ActiveHMI.WatchdogTime[1] := #Param.WatchdogTime[1];
       #previous.WatchdogTime[1] := #Param.WatchdogTime[1];
   END_IF;
END_REGION

REGION Network 18: Confirm Modification / Cancel Modification / Modify Param of WatchdogTime[2] for StopFLT
   IF (#ActiveHMI.WatchdogTime[2] >= 0.0) AND #Modifying.WatchdogTime_StopFLT AND #Confirm THEN
       #Param.WatchdogTime[2] := #ActiveHMI.WatchdogTime[2];
       #previous.WatchdogTime[2] := #ActiveHMI.WatchdogTime[2];
   END_IF;
   IF ((0.0 > #ActiveHMI.WatchdogTime[2]) AND #Modifying.WatchdogTime_StopFLT) OR #Cancel THEN
       #ActiveHMI.WatchdogTime[2] := #Param.WatchdogTime[2];
       #previous.WatchdogTime[2] := #Param.WatchdogTime[2];
   END_IF;
   IF #Param.WatchdogTime[2] <> #previous.WatchdogTime[2] THEN
       #ActiveHMI.WatchdogTime[2] := #Param.WatchdogTime[2];
       #previous.WatchdogTime[2] := #Param.WatchdogTime[2];
   END_IF;
END_REGION

REGION Network 19: Confirm Modification / Cancel Modification / Modify Param of WatchdogTime[3] for FwdFLT
   IF (#ActiveHMI.WatchdogTime[3] >= 0.0) AND #Modifying.WatchdogTime_ForwardFLT AND #Confirm THEN
       #Param.WatchdogTime[3] := #ActiveHMI.WatchdogTime[3];
       #previous.WatchdogTime[3] := #ActiveHMI.WatchdogTime[3];
   END_IF;
   IF ((0.0 > #ActiveHMI.WatchdogTime[3]) AND #Modifying.WatchdogTime_ForwardFLT) OR #Cancel THEN
       #ActiveHMI.WatchdogTime[3] := #Param.WatchdogTime[3];
       #previous.WatchdogTime[3] := #Param.WatchdogTime[3];
   END_IF;
   IF #Param.WatchdogTime[3] <> #previous.WatchdogTime[3] THEN
       #ActiveHMI.WatchdogTime[3] := #Param.WatchdogTime[3];
       #previous.WatchdogTime[3] := #Param.WatchdogTime[3];
   END_IF;
END_REGION

REGION Network 20: Confirm Modification / Cancel Modification / Modify Param of WatchdogTime[4] for RvsFLT
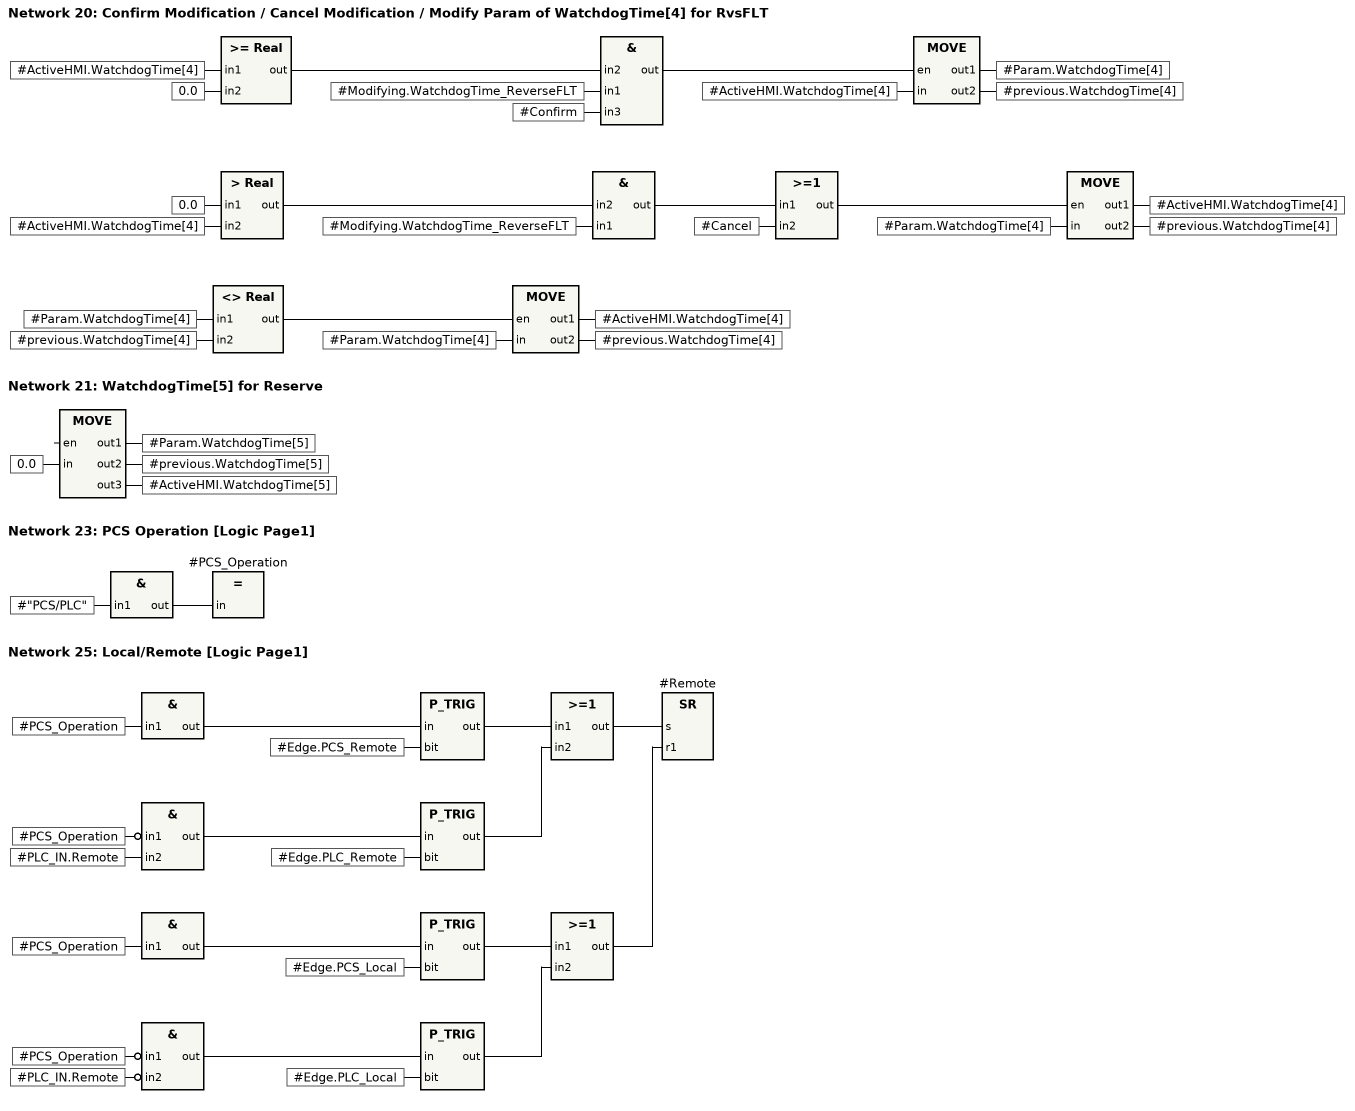
   IF (#ActiveHMI.WatchdogTime[4] >= 0.0) AND #Modifying.WatchdogTime_ReverseFLT AND #Confirm THEN
       #Param.WatchdogTime[4] := #ActiveHMI.WatchdogTime[4];
       #previous.WatchdogTime[4] := #ActiveHMI.WatchdogTime[4];
   END_IF;
   IF ((0.0 > #ActiveHMI.WatchdogTime[4]) AND #Modifying.WatchdogTime_ReverseFLT) OR #Cancel THEN
       #ActiveHMI.WatchdogTime[4] := #Param.WatchdogTime[4];
       #previous.WatchdogTime[4] := #Param.WatchdogTime[4];
   END_IF;
   IF #Param.WatchdogTime[4] <> #previous.WatchdogTime[4] THEN
       #ActiveHMI.WatchdogTime[4] := #Param.WatchdogTime[4];
       #previous.WatchdogTime[4] := #Param.WatchdogTime[4];
   END_IF;
END_REGION

REGION Network 21: WatchdogTime[5] for Reserve
   #Param.WatchdogTime[5] := 0.0;
   #previous.WatchdogTime[5] := 0.0;
   #ActiveHMI.WatchdogTime[5] := 0.0;
END_REGION

REGION Network 22: ----------- Logic Diagram -------------------------------------------------------------------------------------------------------------------------------------------------------------
END_REGION

REGION Network 23: PCS Operation [Logic Page1]
   // PCS_Operation=0 : PLC Operation 
   //  PCS_Operation=1 : PCS Operation
   #PCS_Operation := #"PCS/PLC";
END_REGION

REGION Network 24: Motor Running [Logic Page6]
END_REGION

REGION Network 25: Local/Remote [Logic Page1]
   // Remote=0 : Local(Filed)  /  Remote=1 : Remote
   #_w1 := #PCS_Operation AND NOT #Edge.PCS_Remote;   // rising edge
   #Edge.PCS_Remote := #PCS_Operation;
   #_w2 := NOT #PCS_Operation AND #PLC_IN.Remote;
   #_w3 := #_w2 AND NOT #Edge.PLC_Remote;   // rising edge
   #Edge.PLC_Remote := #_w2;
   #_w4 := #PCS_Operation AND NOT #Edge.PCS_Local;   // rising edge
   #Edge.PCS_Local := #PCS_Operation;
   #_w5 := NOT #PCS_Operation AND NOT #PLC_IN.Remote;
   #_w6 := #_w5 AND NOT #Edge.PLC_Local;   // rising edge
   #Edge.PLC_Local := #_w5;
   IF #_w1 OR #_w3 THEN
       #Remote := TRUE;   // SR flip-flop
   END_IF;
   IF #_w4 OR #_w6 THEN #Remote := FALSE; END_IF;
END_REGION

REGION Network 26: Auto/Manual [Logic Page1]
   // Auto=0 : Manual Mode  /  Auto=1 : Auto Mode
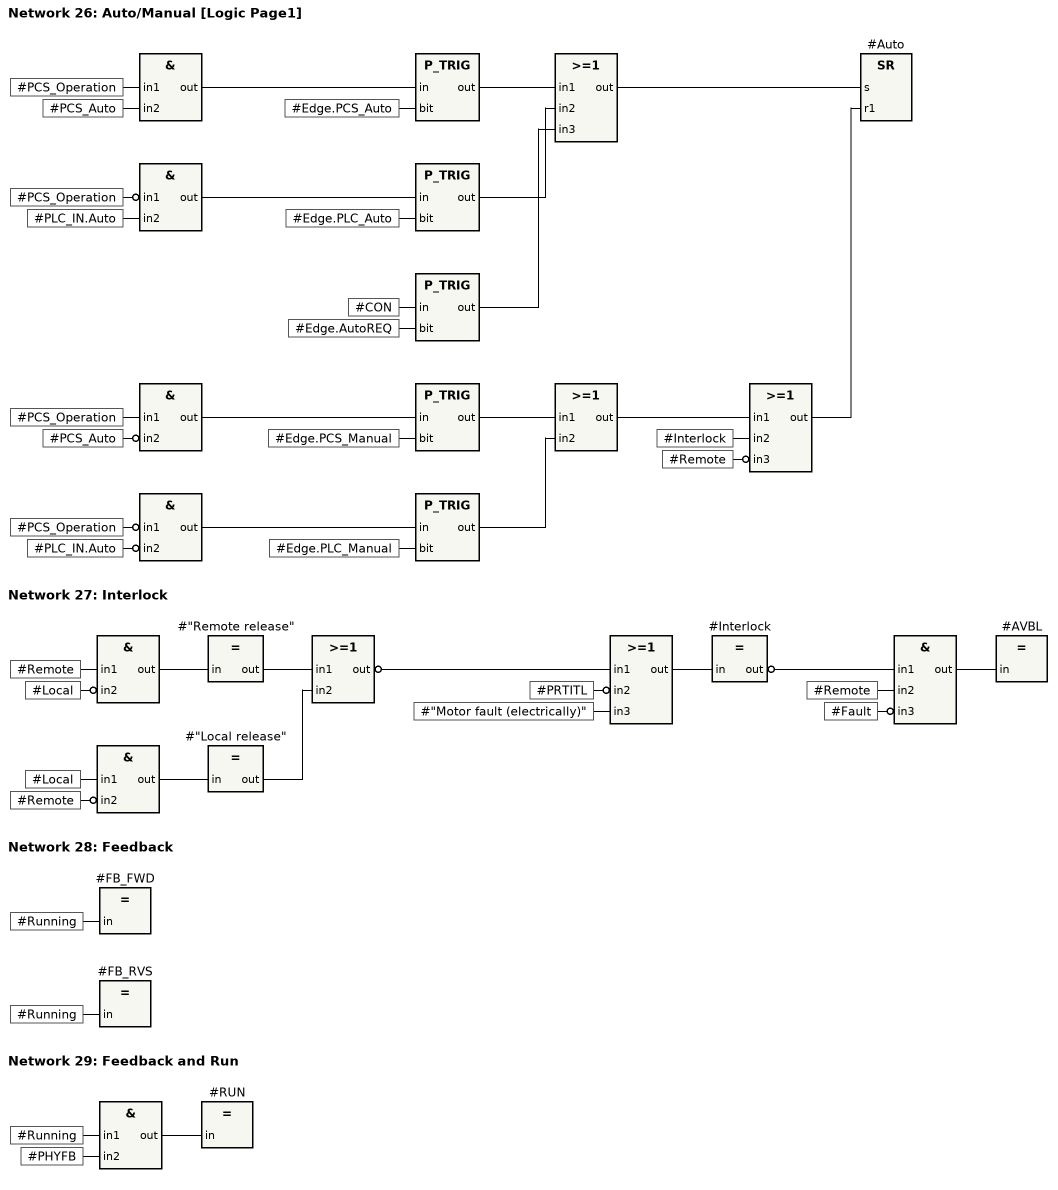
   #_w1 := #PCS_Operation AND #PCS_Auto;
   #_w2 := #_w1 AND NOT #Edge.PCS_Auto;   // rising edge
   #Edge.PCS_Auto := #_w1;
   #_w3 := NOT #PCS_Operation AND #PLC_IN.Auto;
   #_w4 := #_w3 AND NOT #Edge.PLC_Auto;   // rising edge
   #Edge.PLC_Auto := #_w3;
   #_w5 := #CON AND NOT #Edge.AutoREQ;   // rising edge
   #Edge.AutoREQ := #CON;
   #_w6 := #PCS_Operation AND NOT #PCS_Auto;
   #_w7 := #_w6 AND NOT #Edge.PCS_Manual;   // rising edge
   #Edge.PCS_Manual := #_w6;
   #_w8 := NOT #PCS_Operation AND NOT #PLC_IN.Auto;
   #_w9 := #_w8 AND NOT #Edge.PLC_Manual;   // rising edge
   #Edge.PLC_Manual := #_w8;
   IF #_w2 OR #_w4 OR #_w5 THEN
       #Auto := TRUE;   // SR flip-flop
   END_IF;
   IF #_w7 OR #_w9 OR #Interlock OR NOT #Remote THEN #Auto := FALSE; END_IF;
END_REGION

REGION Network 27: Interlock
   #"Remote release" := #Remote AND NOT #Local;
   #"Local release" := #Local AND NOT #Remote;
   #_w1 := NOT (#"Remote release" OR #"Local release") OR NOT #PRTITL OR #"Motor fault (electrically)";
   #Interlock := #_w1;
   #AVBL := NOT #_w1 AND #Remote AND NOT #Fault;
END_REGION

REGION Network 28: Feedback
   #FB_FWD := #Running;
   #FB_RVS := #Running;
END_REGION

REGION Network 29: Feedback and Run
   #RUN := #Running AND #PHYFB;
END_REGION

REGION Network 30: Start Enable [Logic Page4]
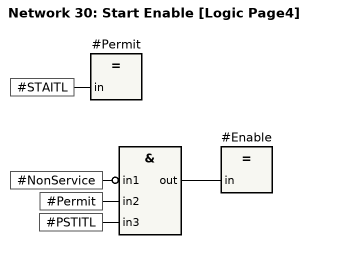
   #Permit := #STAITL;
   #Enable := NOT #NonService AND #Permit AND #PSTITL;
END_REGION

REGION Network 31: Start/Stop [Logic Page4]
   // Start=0(Stop=1) : Motor Stop Requet
   // Start=1(Stop=0) : Motor Start Requet
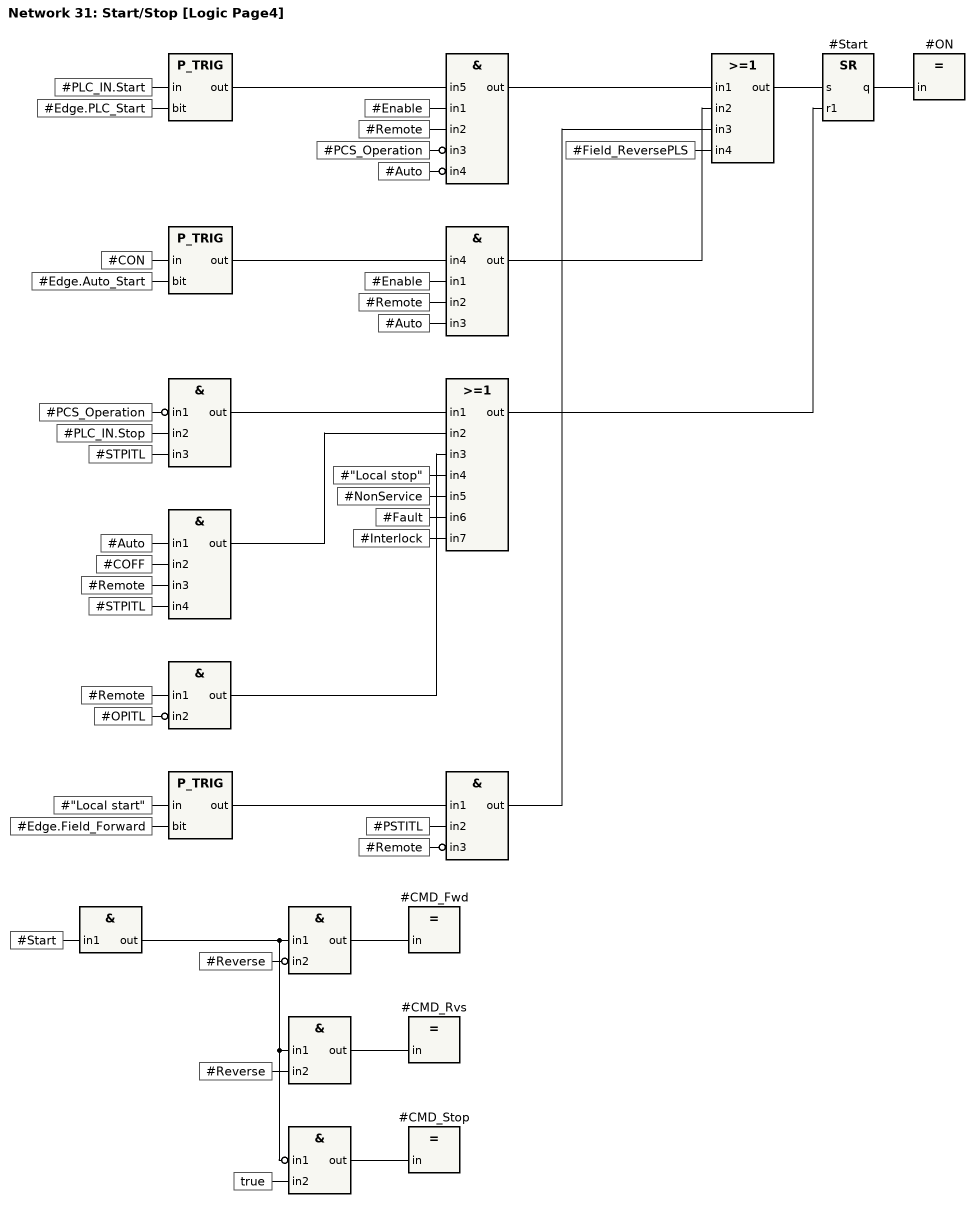
   #_w1 := #PLC_IN.Start AND NOT #Edge.PLC_Start;   // rising edge
   #Edge.PLC_Start := #PLC_IN.Start;
   #_w2 := #CON AND NOT #Edge.Auto_Start;   // rising edge
   #Edge.Auto_Start := #CON;
   #_w3 := #"Local start" AND NOT #Edge.Field_Forward;   // rising edge
   #Edge.Field_Forward := #"Local start";
   IF (#_w1 AND #Enable AND #Remote AND NOT #PCS_Operation AND NOT #Auto) OR (#_w2 AND #Enable AND #Remote AND #Auto) OR (#_w3 AND #PSTITL AND NOT #Remote) OR #Field_ReversePLS THEN
       #Start := TRUE;   // SR flip-flop
   END_IF;
   IF (NOT #PCS_Operation AND #PLC_IN.Stop AND #STPITL) OR (#Auto AND #COFF AND #Remote AND #STPITL) OR (#Remote AND NOT #OPITL) OR #"Local stop" OR #NonService OR #Fault OR #Interlock THEN
       #Start := FALSE;
   END_IF;
   #ON := #Start;
   #CMD_Fwd := #Start AND NOT #Reverse;
   #CMD_Rvs := #Start AND #Reverse;
   #CMD_Stop := NOT #Start AND true;
END_REGION

REGION Network 32: Set PT [Logic Page5]
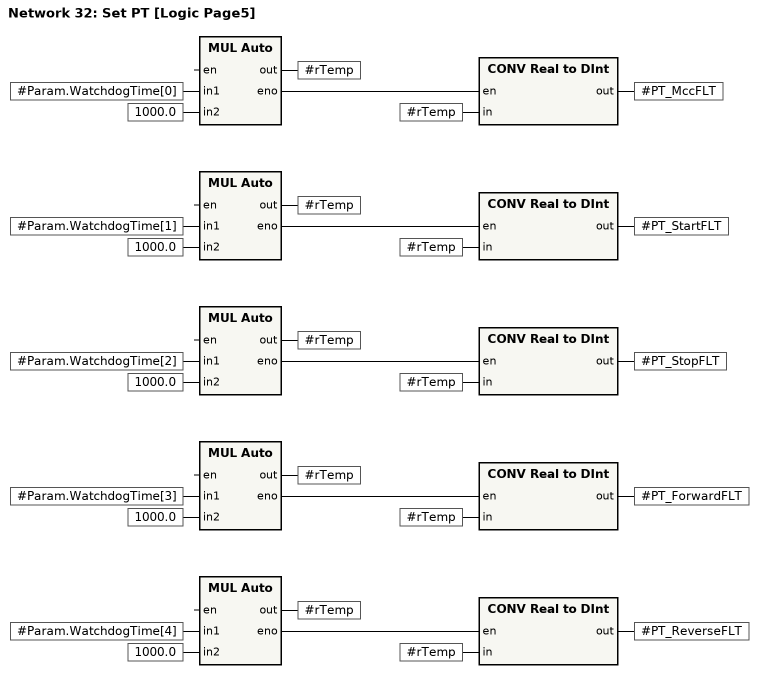
   #rTemp := #Param.WatchdogTime[0] * 1000.0;
   #PT_MccFLT := REAL_TO_DINT(#rTemp);
   #rTemp := #Param.WatchdogTime[1] * 1000.0;
   #PT_StartFLT := REAL_TO_DINT(#rTemp);
   #rTemp := #Param.WatchdogTime[2] * 1000.0;
   #PT_StopFLT := REAL_TO_DINT(#rTemp);
   #rTemp := #Param.WatchdogTime[3] * 1000.0;
   #PT_ForwardFLT := REAL_TO_DINT(#rTemp);
   #rTemp := #Param.WatchdogTime[4] * 1000.0;
   #PT_ReverseFLT := REAL_TO_DINT(#rTemp);
END_REGION

REGION Network 33: Fault [Logic Page5]
   // Fault=1 : Faulty
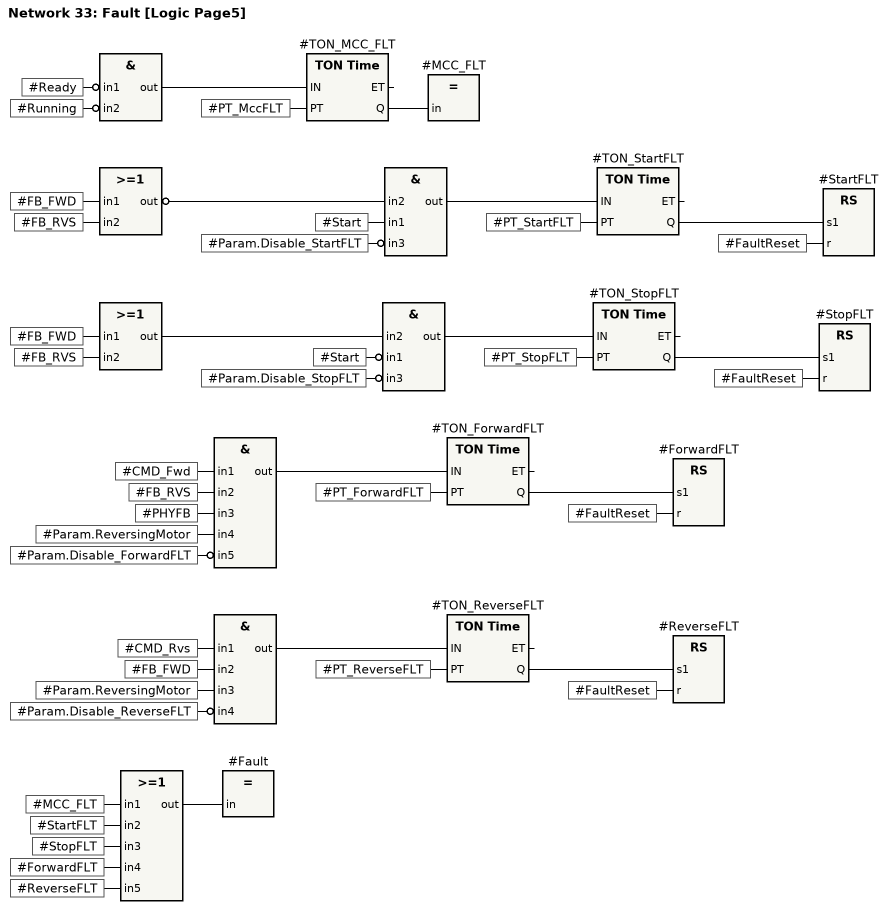
   #TON_MCC_FLT(IN := NOT #Ready AND NOT #Running, PT := #PT_MccFLT);   // TON
   #MCC_FLT := #TON_MCC_FLT.Q;
   #TON_StartFLT(IN := NOT (#FB_FWD OR #FB_RVS) AND #Start AND NOT #Param.Disable_StartFLT, PT := #PT_StartFLT);   // TON
   IF #FaultReset THEN
       #StartFLT := FALSE;   // RS flip-flop
   END_IF;
   IF #TON_StartFLT.Q THEN #StartFLT := TRUE; END_IF;
   #TON_StopFLT(IN := (#FB_FWD OR #FB_RVS) AND NOT #Start AND NOT #Param.Disable_StopFLT, PT := #PT_StopFLT);   // TON
   IF #FaultReset THEN
       #StopFLT := FALSE;   // RS flip-flop
   END_IF;
   IF #TON_StopFLT.Q THEN #StopFLT := TRUE; END_IF;
   #TON_ForwardFLT(IN := #CMD_Fwd AND #FB_RVS AND #PHYFB AND #Param.ReversingMotor AND NOT #Param.Disable_ForwardFLT,   // TON
                   PT := #PT_ForwardFLT);
   IF #FaultReset THEN
       #ForwardFLT := FALSE;   // RS flip-flop
   END_IF;
   IF #TON_ForwardFLT.Q THEN #ForwardFLT := TRUE; END_IF;
   #TON_ReverseFLT(IN := #CMD_Rvs AND #FB_FWD AND #Param.ReversingMotor AND NOT #Param.Disable_ReverseFLT,   // TON
                   PT := #PT_ReverseFLT);
   IF #FaultReset THEN
       #ReverseFLT := FALSE;   // RS flip-flop
   END_IF;
   IF #TON_ReverseFLT.Q THEN #ReverseFLT := TRUE; END_IF;
   #Fault := #MCC_FLT OR #StartFLT OR #StopFLT OR #ForwardFLT OR #ReverseFLT;
END_REGION

REGION Network 34: -------------------- Other -----------------------------------------------------------------------------------------------------------------------------------------------------------------
END_REGION

REGION Network 35: Drive Run Time Calculation (internal Count)
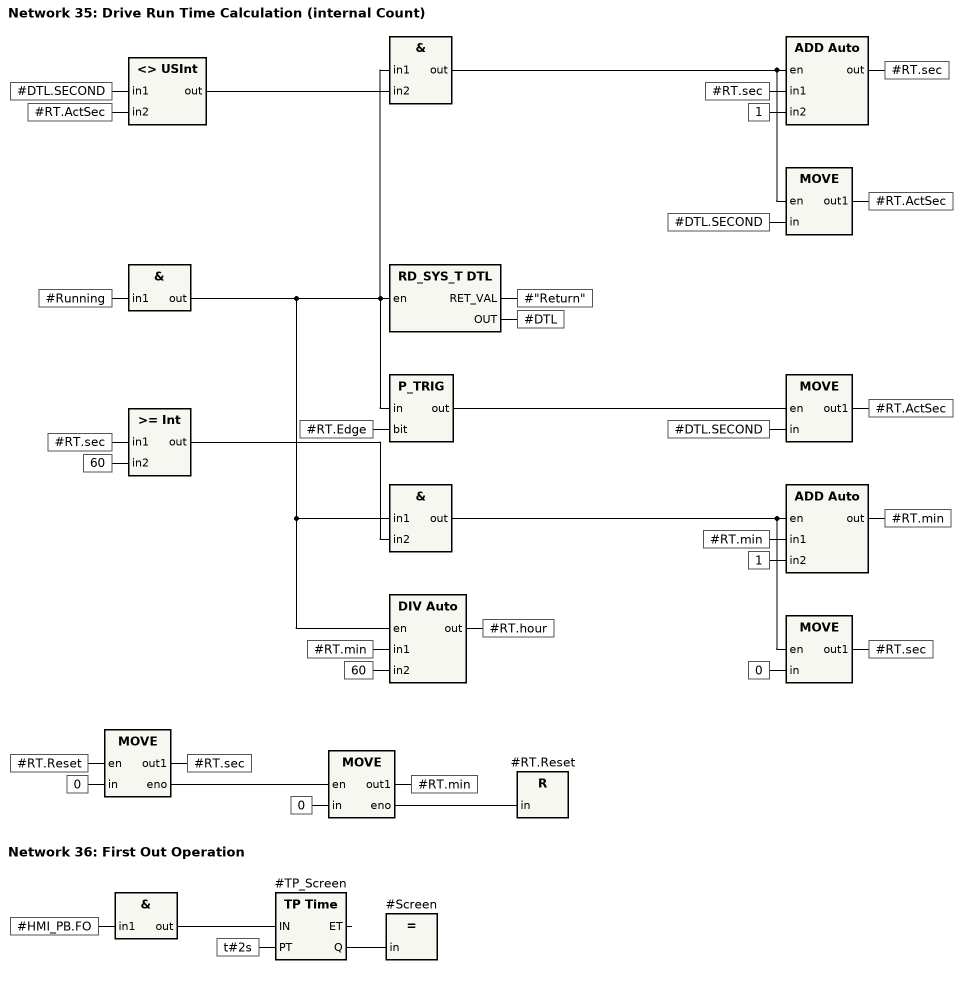
   IF #Running THEN #"Return" := RD_SYS_T(OUT => #DTL); END_IF;
   #_w1 := #Running AND NOT #RT.Edge;   // rising edge
   #RT.Edge := #Running;
   IF #_w1 THEN #RT.ActSec := #DTL.SECOND; END_IF;
   IF #Running AND (#DTL.SECOND <> #RT.ActSec) THEN
       #RT.sec := #RT.sec + 1;
       #RT.ActSec := #DTL.SECOND;
   END_IF;
   IF #Running AND (#RT.sec >= 60) THEN
       #RT.min := #RT.min + 1;
       #RT.sec := 0;
   END_IF;
   IF #Running THEN #RT.hour := #RT.min / 60; END_IF;
   IF #RT.Reset THEN
       #RT.sec := 0;
       #RT.min := 0;
       #RT.Reset := FALSE;
   END_IF;
END_REGION

REGION Network 36: First Out Operation
   #TP_Screen(IN := #HMI_PB.FO, PT := t#2s);   // TP
   #Screen := #TP_Screen.Q;
END_REGION

REGION Network 37: -------------------- HMI Operation(Output) -----------------------------------------------------------------------------------------------------------------------------------
END_REGION

REGION Network 38 (SCL): Set Data to ActiveHMI
   //Drive Run Time 
   #ActiveHMI.RunTime := 0;
END_REGION

REGION Network 39 (SCL): Set Data to Icon
   #icon.Status := #ActiveHMI.Status;
   #icon.Mode := #ActiveHMI.Mode;
   #icon.AlarmCode := #ActiveHMI.AlarmCode;
END_REGION

REGION Network 40 (SCL): Status Code
   // 0 : Unkown
   //  // Case: Forward/Backward is used, Speed1/Speed2 is used
   //    1 : Stop
   //  12 : Stopping Forward 
   //  13 : Starting Forward
   //  15 : Running Forward Speed1
   //  16 : Running Forward Speed2
   //  22 : Stopping Reverse
   //  23: Starting Reverse
   //  25: Running Reverse Speed1
   //  26: Running Reverse Speed2
   //  // Case: Forward/Backward is used, Speed1/Speed2 is not used
   //    1 : Stop
   //  12 : Stopping Forward 
   //  13 : Starting Forward
   //  14: Running Forward
   //  22 : Stopping Reverse
   //  23: Starting Reverse
   //  24: Running Reverse
   //  // Case: Forward/Backward is not used, Speed1/Speed2 is used
   //    1 : Stop
   //    2 : Stopping 
   //    3 : Starting
   //    5 : Running Speed1
   //    6 : Running Speed2
   //  // Case: Forward/Backward is not used, Speed1/Speed2 is not used
   //    1 : Stop
   //    2 : Stopping 
   //    3 : Starting
   //    4: Running
   #ActiveHMI.Status := 0;  // Unknown Status
   // Enable Forward/Reverse, Disable Speed1/Speed2
   IF #Param.ReversingMotor = true AND #Param.SpeedSelect = false THEN
       IF #Ready = TRUE AND #Running = FALSE THEN #ActiveHMI.Status:=1; END_IF; // Stopped
       IF #Running=true AND #Reverse = FALSE THEN #ActiveHMI.Status:=14; END_IF; //Running Forward   
       IF #Running=true AND #Reverse = true THEN #ActiveHMI.Status:=24; END_IF; //Running Reverse
       IF #Start = FALSE AND #Running = TRUE AND #Reverse = false THEN #ActiveHMI.Status:=12; END_IF; // Stopping Forward
       IF #Start = FALSE AND #Running = TRUE AND #Reverse = true THEN #ActiveHMI.Status:=22; END_IF; // Stopping Reverse    
       IF #Start = TRUE AND #Running = FALSE AND #Reverse=false THEN #ActiveHMI.Status:=13; END_IF; // Starting Forward
       IF #Start = TRUE AND #Running = FALSE AND  #Reverse=true THEN #ActiveHMI.Status:=23; END_IF; // Starting Reverse
   END_IF;
   // Disable Forward/Reverse, Disable Speed1/Speed2
   IF #Param.ReversingMotor = false AND #Param.SpeedSelect = false THEN
       IF #Ready = TRUE AND #Running = FALSE THEN #ActiveHMI.Status:=1; END_IF; // Stopped
       IF #Running = TRUE THEN #ActiveHMI.Status:=4; END_IF; //Running   
       IF #Start = FALSE AND #Running = TRUE  THEN #ActiveHMI.Status:=2; END_IF; // Stopping Forward
       IF #Start = TRUE AND #Running = FALSE THEN #ActiveHMI.Status:=3; END_IF; // Starting Forward
   END_IF;
END_REGION

REGION Network 41 (SCL): Mode
   // Mode=1 : Manual Start/Stop by Local(Field) : Charactor 'L' on HMI
   // Mode=2 : Operation by PCS : Charactor 'P' on HMI
   // Mode=3 : Operation by PLC(HMI) : Charactor 'R' on HMI
   // Mode=4 : Auto Control : Charactor 'A' on HMI
   IF #Remote=false THEN
       #ActiveHMI.Mode:=1;  // Loal Operation --> Display 'L'
   ELSIF #PCS_Operation=true AND #Remote=true AND #Auto=false THEN
       #ActiveHMI.Mode:=2; ; // PCS&Remote&Mamual = PCS Manual Operation  --> Display 'P'
   ELSIF #PCS_Operation=false AND #Remote=true AND #Auto=false THEN
       #ActiveHMI.Mode:=3;; // PLC&Remote&Manual = PLC Manual Operation --> Display 'R'
   ELSIF #Auto=true THEN
       #ActiveHMI.Mode:=4;  // PCS&Remote&Auto = Auto Operation --> Display 'A'
   ELSE
       #ActiveHMI.Mode := 0;
   END_IF;
END_REGION

REGION Network 42 (SCL): Alarm Code
   // 0 : No Alarm
   // 200 : Not Permitted
   // 400 : Interlocked
   // 410 : Not Serviced
   // 420 : MCC Fault
   IF #Permit = true AND #Interlock = false AND #NonService = false AND #Fault = false THEN
       #ActiveHMI.AlarmCode := 0; // No Alarm
   END_IF;
   IF #Permit= false THEN #ActiveHMI.AlarmCode := 200; END_IF;  // Permit
   IF #Interlock=true THEN #ActiveHMI.AlarmCode := 400; END_IF;  // Interlock
   IF #NonService=true THEN #ActiveHMI.AlarmCode := 410; END_IF; // Not Serviced
   IF #Fault=true THEN #ActiveHMI.AlarmCode:=420; END_IF;  // MCC(External) Fault
END_REGION

REGION Network 43 (SCL): Object Control on Active HMI (Operation Enabled HMI)
   // 0 : Invisible
   //   1 : Display PB, Dark Color, modification is allowed
   //   2 : Display PB, Flashing, modification is allowed
   //   4 : Display PB, Light color, modification is allowed
   //   11 : Display PB, Dark Color, modification is not allowed
   //   12 : Display PB, Flashing, modification is not allowed
   //   14 : Display PB, Light color, modification is not allowed
   //   21 : Display Status, Dark Color
   //   22 : Display Status, Flashing
   //   24 : Display Status, Light color
   IF #PopupCtrl.Opened=true THEN

       // Status Area
       // Ojbject[0]/[1] : PCS/PLC
       IF #PCS_Operation=true THEN #ActiveHMI.Object[0]:=24; ELSE #ActiveHMI.Object[0]:=21; END_IF;
       IF #PCS_Operation=true THEN #ActiveHMI.Object[1]:=21; ELSE #ActiveHMI.Object[1]:=24; END_IF;
       // Ojbject[2] : Fail
       IF #Fault=true THEN  #ActiveHMI.Object[2]:=24; ELSE #ActiveHMI.Object[2]:=21; END_IF;
       // Ojbject[3] : Interlock
       IF #Interlock=true THEN #ActiveHMI.Object[3]:=24; ELSE #ActiveHMI.Object[3]:=21; END_IF;
       // Ojbject[4] : Service
       IF #NonService=false THEN #ActiveHMI.Object[4]:=24; ELSE #ActiveHMI.Object[4]:=21; END_IF;
       // Ojbject[5] : Permit
       IF #Permit=true THEN #ActiveHMI.Object[5]:=24; ELSE #ActiveHMI.Object[5]:=21; END_IF;
       // Ojbject[6]/[7] : Start/Stop
       #ActiveHMI.Object[6]:=21;
       #ActiveHMI.Object[7]:=21;
       IF #Ready = TRUE AND #Running = FALSE THEN
           #ActiveHMI.Object[6]:=21;
           #ActiveHMI.Object[7]:=24;
       END_IF;
       IF #Running = true THEN
           #ActiveHMI.Object[6]:=24;
           #ActiveHMI.Object[7]:=21;
       END_IF;
       IF #Start = TRUE AND #Running = FALSE THEN
           #ActiveHMI.Object[6]:=22;
           #ActiveHMI.Object[7]:=21;
       END_IF;
       IF #Start = FALSE AND #Running = TRUE THEN
           #ActiveHMI.Object[6]:=21;
           #ActiveHMI.Object[7]:=22;
       END_IF;
       // Object[8] : FO
       IF #FO=true THEN #ActiveHMI.Object[8]:=4; ELSE #ActiveHMI.Object[8]:=1; END_IF;
       // Object[9] : Reserve
       #ActiveHMI.Object[9]:=1;

       // Mode Area
       //Object[10]/[11] : Remote/Local
       IF #PCS_Operation=false THEN
           IF #Remote=true THEN #ActiveHMI.Object[10]:=14; ELSE #ActiveHMI.Object[10]:=1; END_IF;
           IF #Remote=true THEN #ActiveHMI.Object[11]:=1; ELSE #ActiveHMI.Object[11]:=14; END_IF;
       ELSE
           IF #Remote=true THEN #ActiveHMI.Object[10]:=24; ELSE #ActiveHMI.Object[10]:=21; END_IF;
           IF #Remote=true THEN #ActiveHMI.Object[11]:=21; ELSE #ActiveHMI.Object[11]:=24; END_IF;
       END_IF;
       //Object[12]/[13] : Auto/Manual
       IF #PCS_Operation=false AND #Remote=true AND #Interlock=false THEN
           IF #Auto=true THEN #ActiveHMI.Object[12]:=14; ELSE #ActiveHMI.Object[12]:=1; END_IF;
           IF #Auto=true THEN #ActiveHMI.Object[13]:=1; ELSE #ActiveHMI.Object[13]:=14; END_IF;
       ELSE
           IF #Auto=true THEN #ActiveHMI.Object[12]:=24; ELSE #ActiveHMI.Object[12]:=21; END_IF;
           IF #Auto=true THEN #ActiveHMI.Object[13]:=21; ELSE #ActiveHMI.Object[13]:=24; END_IF;
       END_IF;
       //Object[14]/[15] : Forward/Reverse
       IF #Param.ReversingMotor=true THEN
           IF #PCS_Operation=false AND #Remote=true AND #Auto=false THEN
               IF #Reverse=true THEN
                   IF #Start=false THEN #ActiveHMI.Object[14]:=1; ELSE #ActiveHMI.Object[14]:=11; END_IF;
                   #ActiveHMI.Object[15]:=14;
               ELSE
                   #ActiveHMI.Object[14]:=14;
                   IF #Start=false THEN #ActiveHMI.Object[15]:=1; ELSE #ActiveHMI.Object[15]:=11; END_IF;
               END_IF;
           ELSE
               IF #Reverse=true THEN #ActiveHMI.Object[14]:=21; ELSE #ActiveHMI.Object[14]:=24; END_IF;
               IF #Reverse=true THEN #ActiveHMI.Object[15]:=24; ELSE #ActiveHMI.Object[15]:=21; END_IF;
           END_IF;
       ELSE
           #ActiveHMI.Object[14]:=0;
           #ActiveHMI.Object[15]:=0;
       END_IF;
       //Object[16]/[17] : Speed1/Speed2 when ReversingMotor=True
       IF #Param.SpeedSelect=true AND #Param.ReversingMotor=true THEN
           IF #PCS_Operation=false AND #Remote=true AND #Auto=false THEN
               IF #Speed=true THEN
                   IF #Start=false THEN #ActiveHMI.Object[16]:=1; ELSE #ActiveHMI.Object[16]:=11; END_IF;
                   #ActiveHMI.Object[17] := 14;
               ELSE
                   #ActiveHMI.Object[16] := 14;
                   IF #Start=false THEN #ActiveHMI.Object[17]:=1; ELSE #ActiveHMI.Object[17]:=11; END_IF;
               END_IF;
           ELSE
               IF #Speed=true THEN #ActiveHMI.Object[16]:=21; ELSE #ActiveHMI.Object[16]:=24; END_IF;
               IF #Speed=true THEN #ActiveHMI.Object[17]:=24; ELSE #ActiveHMI.Object[17]:=21; END_IF;
           END_IF;
       ELSE
           #ActiveHMI.Object[16] := 0;
           #ActiveHMI.Object[17] := 0;
       END_IF;
       //Object[18]/[19] : Speed1b/Speed2b when ReversingMotor=False
       IF #Param.SpeedSelect=true AND #Param.ReversingMotor=false THEN
           IF #PCS_Operation=false AND #Remote=true AND #Auto=false THEN
               IF #Speed=true THEN
                   IF #Start=false THEN #ActiveHMI.Object[18]:=1; ELSE #ActiveHMI.Object[18]:=11; END_IF;
                   #ActiveHMI.Object[19] := 14;
               ELSE
                   #ActiveHMI.Object[18] := 14;
                   IF #Start=false THEN #ActiveHMI.Object[19]:=1; ELSE #ActiveHMI.Object[19]:=11; END_IF;
               END_IF;
           ELSE
               IF #Speed=true THEN #ActiveHMI.Object[18]:=21; ELSE #ActiveHMI.Object[18]:=24; END_IF;
               IF #Speed=true THEN #ActiveHMI.Object[19]:=24; ELSE #ActiveHMI.Object[19]:=21; END_IF;
           END_IF;
       ELSE
           #ActiveHMI.Object[18] := 0;
           #ActiveHMI.Object[19] := 0;
       END_IF;

       // Manual Operation Area
       //Object [20]/[21] : Start/Stop
       IF #PCS_Operation=false AND #Remote=true AND #Auto=false THEN
           IF #Start=true THEN #ActiveHMI.Object[20]:=14; ELSE #ActiveHMI.Object[20]:=1; END_IF;
           IF #Start=true THEN #ActiveHMI.Object[21]:=1; ELSE #ActiveHMI.Object[21]:=14; END_IF;
       ELSE
           IF #Start=true THEN #ActiveHMI.Object[20]:=24; ELSE #ActiveHMI.Object[20]:=21; END_IF;
           IF #Start=true THEN #ActiveHMI.Object[21]:=21; ELSE #ActiveHMI.Object[21]:=24; END_IF;
       END_IF;

       //Object [22]-[26] : Watchdog Time
       #ActiveHMI.Object[22] := 0;
       IF #Modifying.WatchdogTime_StartFLT=true THEN #ActiveHMI.Object[23]:=2; ELSE #ActiveHMI.Object[23]:=4; END_IF;
       IF #Modifying.WatchdogTime_StopFLT=true THEN #ActiveHMI.Object[24]:=2; ELSE #ActiveHMI.Object[24]:=4; END_IF;
       IF #Modifying.WatchdogTime_ForwardFLT=true THEN #ActiveHMI.Object[25]:=2; ELSE #ActiveHMI.Object[25]:=4; END_IF;
       IF #Modifying.WatchdogTime_ReverseFLT=true THEN #ActiveHMI.Object[26]:=2; ELSE #ActiveHMI.Object[26]:=4; END_IF;

   END_IF;
END_REGION

REGION Network 44 (SCL): Object Control on Passive HMI (Operation Disabled HMI)
   // 0 : Invisible
   //   1 : Display PB, Dark Color, modification is allowed
   //   2 : Display PB, Flashing, modification is allowed
   //   4 : Display PB, Light color, modification is allowed
   //   11 : Display PB, Dark Color, modification is not allowed
   //   12 : Display PB, Flashing, modification is not allowed
   //   14 : Display PB, Light color, modification is not allowed
   //   21 : Display Status, Dark Color
   //   22 : Display Status, Flashing
   //   24 : Display Status, Light color
    // Status Area
       // Ojbject[0]/[1] : PCS/PLC
       IF #PCS_Operation=true THEN #PassiveHMI.Object[0]:=24; ELSE #PassiveHMI.Object[0]:=21; END_IF;
       IF #PCS_Operation=true THEN #PassiveHMI.Object[1]:=21; ELSE #PassiveHMI.Object[1]:=24; END_IF;
       // Ojbject[2] : Fail
       IF #Fault=true THEN #PassiveHMI.Object[2]:=24; ELSE #PassiveHMI.Object[2]:=21; END_IF;
       // Ojbject[3] : Interlock
       IF #Interlock=true THEN #PassiveHMI.Object[3]:=24; ELSE #PassiveHMI.Object[3]:=21; END_IF;
       // Ojbject[4] : Service
       IF #NonService=false THEN #PassiveHMI.Object[4]:=24; ELSE #PassiveHMI.Object[4]:=21; END_IF;
       // Ojbject[5] : Permit
       IF #Permit=true THEN #PassiveHMI.Object[5]:=24; ELSE #PassiveHMI.Object[5]:=21; END_IF;
       // Ojbject[6]/[7] : Start/Stop
       #PassiveHMI.Object[6]:=21;
       #PassiveHMI.Object[7]:=21;
       IF #Ready = TRUE AND #Running = FALSE THEN
           #PassiveHMI.Object[6]:=21;
           #PassiveHMI.Object[7]:=24;
       END_IF;
       IF #Running=true THEN
           #PassiveHMI.Object[6]:=24;
           #PassiveHMI.Object[7]:=21;
       END_IF;
       IF #Start = TRUE AND #Running = FALSE THEN
           #PassiveHMI.Object[6]:=22;
           #PassiveHMI.Object[7]:=21;
       END_IF;
       IF #Start = FALSE AND #Running = TRUE THEN
           #PassiveHMI.Object[6]:=21;
           #PassiveHMI.Object[7]:=22;
       END_IF;
       // Object[8] : FO
       IF #FO=true THEN #PassiveHMI.Object[8]:=4; ELSE #PassiveHMI.Object[8]:=1; END_IF;
       // Object[9] : Reserve

       // Mode Area
       //Object[10]/[11] : Remote/Local
       IF #PCS_Operation=true THEN
           IF #Remote=true THEN #PassiveHMI.Object[10]:=24; ELSE #PassiveHMI.Object[10]:=21; END_IF;
           IF #Remote=true THEN #PassiveHMI.Object[11]:=21; ELSE #PassiveHMI.Object[11]:=24; END_IF;
       ELSE
           IF #Remote=true THEN #PassiveHMI.Object[10]:=14; ELSE #PassiveHMI.Object[10]:=11; END_IF;
           IF #Remote=true THEN #PassiveHMI.Object[11]:=11; ELSE #PassiveHMI.Object[11]:=14; END_IF;
       END_IF;
       //Object[12]/[13] : Auto/Manual
       IF #PCS_Operation=true OR #Remote=false THEN
           IF #Auto=true THEN #PassiveHMI.Object[12]:=24; ELSE #PassiveHMI.Object[12]:=21; END_IF;
           IF #Auto=true THEN #PassiveHMI.Object[13]:=21; ELSE #PassiveHMI.Object[13]:=24; END_IF;
       ELSE
           IF #Auto=true THEN #PassiveHMI.Object[12]:=14; ELSE #PassiveHMI.Object[12]:=11; END_IF;
           IF #Auto=true THEN #PassiveHMI.Object[13]:=11; ELSE #PassiveHMI.Object[13]:=14; END_IF;
       END_IF;
       //Object[14]/[15] : Forward/Reverse
       IF #Param.ReversingMotor=true THEN
           IF #PCS_Operation=true OR #Remote=false AND #Auto=false THEN
               IF #Reverse=true THEN #PassiveHMI.Object[14]:=21; ELSE #PassiveHMI.Object[14]:=24; END_IF;
               IF #Reverse=true THEN #PassiveHMI.Object[15]:=24; ELSE #PassiveHMI.Object[15]:=21; END_IF;
           ELSE
               IF #Reverse=true THEN #PassiveHMI.Object[14]:=11; ELSE #PassiveHMI.Object[14]:=14; END_IF;
               IF #Reverse=true THEN #PassiveHMI.Object[15]:=14; ELSE #PassiveHMI.Object[15]:=11; END_IF;
           END_IF;
       ELSE
           #PassiveHMI.Object[14]:=0;
           #PassiveHMI.Object[15]:=0;
       END_IF;
       //Object[16]/[17] : Speed1/Speed2
       IF #Param.SpeedSelect=true AND #Param.ReversingMotor=true THEN
           IF #PCS_Operation=true OR #Remote=false AND #Auto=false THEN
               IF #Speed=true THEN #PassiveHMI.Object[16]:=21; ELSE #PassiveHMI.Object[16]:=24; END_IF;
               IF #Speed=true THEN #PassiveHMI.Object[17]:=24; ELSE #PassiveHMI.Object[17]:=21; END_IF;
           ELSE
               IF #Speed=true THEN #PassiveHMI.Object[16]:=11; ELSE #PassiveHMI.Object[16]:=14; END_IF;
               IF #Speed=true THEN #PassiveHMI.Object[17]:=14; ELSE #PassiveHMI.Object[17]:=11; END_IF;
           END_IF;
       ELSE
           #PassiveHMI.Object[16]:=0;
           #PassiveHMI.Object[17]:=0;
       END_IF;
       //Object [18]/[19] : Speed1b/Speed2b
       IF #Param.SpeedSelect=true AND #Param.ReversingMotor=false THEN
           IF #PCS_Operation=true OR #Remote=false AND #Auto=false THEN
               IF #Speed=true THEN #PassiveHMI.Object[18]:=21; ELSE #PassiveHMI.Object[18]:=24; END_IF;
               IF #Speed=true THEN #PassiveHMI.Object[19]:=24; ELSE #PassiveHMI.Object[19]:=21; END_IF;
           ELSE
               IF #Speed=true THEN #PassiveHMI.Object[18]:=11; ELSE #PassiveHMI.Object[18]:=14; END_IF;
               IF #Speed=true THEN #PassiveHMI.Object[19]:=14; ELSE #PassiveHMI.Object[19]:=11; END_IF;
           END_IF;
       ELSE
           #PassiveHMI.Object[18] := 0;
           #PassiveHMI.Object[19] := 0;
       END_IF;
       // Manual Operation Area
       //Object [20]/[21] : Start/Stop
       IF #PCS_Operation=true OR #Remote=false AND #Auto=false THEN
           IF #Running=true THEN #PassiveHMI.Object[20]:=24; ELSE #PassiveHMI.Object[20]:=21; END_IF;
           IF #Running=true THEN #PassiveHMI.Object[21]:=21; ELSE #PassiveHMI.Object[21]:=24; END_IF;
       ELSE
           IF #Running=true THEN #PassiveHMI.Object[20]:=14; ELSE #PassiveHMI.Object[20]:=11; END_IF;
           IF #Running=true THEN #PassiveHMI.Object[21]:=11; ELSE #PassiveHMI.Object[21]:=14; END_IF;
       END_IF;

       //Object [22]-[26] : Watchdog Time
       #PassiveHMI.Object[22] := 0;
       #PassiveHMI.Object[23] := 11;
       #PassiveHMI.Object[24] := 11;
       #PassiveHMI.Object[25] := 11;
       #PassiveHMI.Object[26] := 11;
END_REGION

REGION Network 45 (SCL): Send Data to HMI (Only for display on HMI and No operatin is allowed.)
   // Tag Name
   #HMI.TagName := #TagName;
   #HMI.TagComment := #TagComment;
   // Data on base screen
   #HMI.Status := #ActiveHMI.Status;
   #HMI.Mode := #ActiveHMI.Mode;
   #HMI.AlarmCode := #ActiveHMI.AlarmCode;
   // Data on opration screen 
   #HMI.RunTime := #ActiveHMI.RunTime;
   #HMI.WatchdogTime := #ActiveHMI.WatchdogTime;
   #HMI.AnalogValue := #ActiveHMI.AnalogValue;
   // Object
   #HMI.Object := #PassiveHMI.Object;
END_REGION

REGION Network 46 (SCL): Send Popup Screen Data to each HMI
   //Data to HMI
    IF #Popup.TagName=#TagName THEN

           // Data on base screen
           #Popup.Status := #ActiveHMI.Status;
           #Popup.AlarmCode := #ActiveHMI.AlarmCode;
           // Data on opration screen
           #Popup.TagComment := #TagComment;
           #Popup.AnalogValue := #ActiveHMI.AnalogValue;
           #Popup.RunTime := #ActiveHMI.RunTime;
           // PBNo & Object
           IF #PopupCtrl.Activate=true THEN  // Operating by this Popup
               IF #ActiveHMI.PBNo <> #Popup.PBNo THEN
                   #Popup.PBNo := #ActiveHMI.PBNo;
               END_IF;
               #Popup.Object := #ActiveHMI.Object;
               #PopupCtrl.OperationBlocked := false;
           ELSIF #PopupCtrl.Activate=true AND #PopupCtrl.Activate=false THEN  // Opeating by otherPopup
               IF #Popup.PBNo <> -1 THEN
                   #Popup.PBNo := -1;
               END_IF;
               #Popup.Object := #PassiveHMI.Object;
               #PopupCtrl.OperationBlocked := true;
           ELSIF #PopupCtrl.Activate=false AND #PopupCtrl.Activate=false THEN  // Operating by No PopupI
               IF #Popup.PBNo <> 0 THEN
                   #Popup.PBNo := 0;
               END_IF;
               #Popup.Object := #ActiveHMI.Object;
               #PopupCtrl.OperationBlocked := false;
           END_IF;

   END_IF;
END_REGION

REGION Network 47: ----------- END --------------------------------------------------------------------------------------------------------------------------------------------------------------------------------
END_REGION

REGION Network 48 (SCL): ENO
   // ENO=1 when No Fault.
   IF #ActiveHMI.AlarmCode=0 THEN ENO:=true; ELSE ENO:=false; END_IF;
END_REGION
END_FUNCTION_BLOCK
